           in_Anlage_ein            := #iSystemActive,
           in_Quitt_Stoerung        := #aFBRotaryValve,
           in_Ansteuerung_Motor     := #RotaryFeeder.auto_mode_control,
           in_Eingang_Motor         := #iFBRotaryFeeder_on,
           io_Ausgang_Motor         := #qRotaryValve_on,
           io_Motor_in_Betrieb      := #RotaryFeeder.motor_in_operation,
           io_Stoerung              := #fFBRotaryFeeder,
           io_Motorstruktur         := #RotaryFeeder);
NETWORK
TITLE = Discharging: release filter
      A     #SEQUENCE.Discharging.AUTO;
      A     #SEQUENCE.Discharging.RELEASE;
      A     #RotaryFeeder.motor_in_operation;
      AN    #PurgedFilter.auto_mode_control_clock1;
      =     #PurgedFilter.auto_mode_control_clock2;
NETWORK
TITLE = Air purge filter object
      CALL  "FC23 Valve 1-10O" (
           in_Handbedienung_erlaubt := TRUE,
           in_Anlage_ein            := #iSystemActive,
           in_Ansteuerung_Ventil_T1 := #PurgedFilter.auto_mode_control_clock1,
           in_Ansteuerung_Ventil_T2 := #PurgedFilter.auto_mode_control_clock2,
           io_Ausgang_Ventil_1      := #qPurgingFilterV1_on,
           io_Ausgang_Ventil_2      := #qPurgingFilterV2_on,
           io_Ausgang_Ventil_3      := #qPurgingFilterV3_on,
           io_Ausgang_Ventil_4      := #PurgedFilter.quit_valve_5,
           io_Ausgang_Ventil_5      := #PurgedFilter.quit_valve_5,
           io_Ausgang_Ventil_6      := #PurgedFilter.quit_valve_6,
           io_Ausgang_Ventil_7      := #PurgedFilter.quit_valve_7,
           io_Ausgang_Ventil_8      := #PurgedFilter.quit_valve_8,
           io_Ausgang_Ventil_9      := #PurgedFilter.quit_valve_9,
           io_Ausgang_Ventil_10     := #PurgedFilter.quit_valve_10,
           io_Ventil_in_Betrieb     := #PurgedFilter.valve_in_operation,
           io_Ventilstruktur        := #PurgedFilter);
NETWORK
TITLE = Discharging: DISCHARGING ACTIVE
      A     #SEQUENCE.Discharging.RELEASE;
      A     #RotaryFeeder.motor_in_operation;
      A     #Screener.motor_in_operation;
      A     #MetalSeparator.motor_in_operation;
      =     #SEQUENCE.Discharging.ACTIVE;
NETWORK
TITLE = -----------PFCs---------------
NETWORK
TITLE = PFCs: PFC to packing Machine
      A     #SEQUENCE.Discharging.ACTIVE;	// system is ON + feeding is started
      AN    #fRepRotaryValve;
      AN    #fRepScreener;
      AN    #fRepMetalSeparator;
      AN    #fFBRotaryFeeder;
      AN    #fFBScreener;
      AN    #fFBMetalSeparator;
      AN    #fSafetyRotaryFeeder;
      AN    #fToolKeyControl;
      AN    #fSafetyMS;
      AN    #fREC01HighLevel;
      =     #qPFCPM_Active;
      O     #INTERNAL.Flags.StatusHP03.HP03_material_signal;
      O     #INTERNAL.Flags.StatusREC01.REC01_material_signal;
      =     #qPFCPM_Product;
NETWORK
TITLE = ---------Statuses to HMI----------------
NETWORK
TITLE = Status to HMI: Filling STATUS
      AN    #SEQUENCE.Filling.RELEASE;
      AN    #SEQUENCE.Filling.ACTIVE;
      JCN   FRA;	// status release assignment
      L     0;
      JU    FAF;	// status assignmnet is finished 
FRA:  A     #SEQUENCE.Filling.RELEASE;
      AN    #SEQUENCE.Filling.ACTIVE;
      JCN   FAA;	// status active 
      L     1;
      JU    FAF;
FAA:  A     #SEQUENCE.Filling.RELEASE;
      A     #SEQUENCE.Filling.ACTIVE;
      L     2;
FAF:  T     #HMI.PV.StatusProcessFilling;
NETWORK
TITLE = Status to HMI: Discharging STATUS
      AN    #SEQUENCE.Discharging.RELEASE;
      AN    #SEQUENCE.Discharging.ACTIVE;
      JCN   DRA;	// status release assignment
      L     0;
      JU    DAF;	// status assignmnet is finished 
DRA:  A     #SEQUENCE.Discharging.RELEASE;
      AN    #SEQUENCE.Discharging.ACTIVE;
      JCN   DAA;	// status active 
      L     1;
      JU    DAF;
DAA:  A     #SEQUENCE.Discharging.RELEASE;
      A     #SEQUENCE.Discharging.ACTIVE;
      L     2;
DAF:  T     #HMI.PV.StatusProcessDischarging;
NETWORK
TITLE = Statuses to HMI for REC01 and HP03 
      A     #INTERNAL.Flags.StatusREC01.REC01_empty;
      =     #HMI.STATE.REC01_empty;
      A     #INTERNAL.Flags.StatusREC01.REC01_full;
      =     #HMI.STATE.REC01_full;
      A     #INTERNAL.Flags.StatusREC01.REC01_material_signal;
      =     #HMI.STATE.REC01_material_signal;
      A     #INTERNAL.Flags.StatusHP03.HP03_empty;
      =     #HMI.STATE.HP03_empty;
      A     #INTERNAL.Flags.StatusHP03.HP03_full;
      =     #HMI.STATE.HP03_full;
      A     #INTERNAL.Flags.StatusHP03.HP03_material_signal;
      =     #HMI.STATE.HP03_material_signal;
NETWORK
TITLE = Status to HMI: PFC to/from Rovema 
//from Rovema
      A     #iPFCPM_Ready;
      =     #HMI.STATE.FROMRovemaReady;
      A     #iPFCPM_TakeProduct;
      =     #HMI.STATE.FROMRovemaTakeMaterial;
// to Rovema
      A     #qPFCPM_Product;
      =     #HMI.STATE.TORovemaProductHP03;
      A     #qPFCPM_Active;
      =     #HMI.STATE.TORovemaActive;
NETWORK
TITLE = ------------Resetting----------------
NETWORK
TITLE = Reset Storage Location
      O     #INTERNAL.Flags.ReleaseFeeding;
      O     #INTERNAL.Flags.StatusREC01.REC01_material_signal;
      O     #INTERNAL.Flags.StatusHP03.HP03_material_signal;
      ON    #iSystemActive;
      FP    #INTERNAL.Flags.FP_StorageLocReset.helpBit;
      =     #INTERNAL.Flags.FP_StorageLocReset.pulseBit;
      A     #INTERNAL.Flags.FP_StorageLocReset.pulseBit;
      JCN   NRS;	//no reset storage
      L     0;
      T     #HMI.PARAM.StorageLocation;
NRS:  NOP   0;
NETWORK
TITLE = ---- interface ----
NETWORK
TITLE = Storage location
      A     #iSystemActive;
      A     #INTERNAL.IF.Silo.SiloNr_correct;
      JCN   NCS;	// correst silo number
      L     #HMI.PV.StorageLocation;
      L     1000;
      +I;
      T     #INTERNAL.IF.Silo.StorageLocation_DB;
      L     200;
      T     #INTERNAL.IF.Silo.StorageLocation_DW;
      CALL  "FC40 copy Obj-IF Master" (
           i_Freigabe               := #IF_Silo.CONTROL.CMD.Request,
           i_Ziel_DB                := #INTERNAL.IF.Silo.StorageLocation_DB,
           i_Ziel_DW                := #INTERNAL.IF.Silo.StorageLocation_DW,
           i_SST_von_Ziel           := #IF_Silo.STATUS,
           i_SST_an_Ziel            := #IF_Silo.CONTROL,
           Ziel_frei                := #INTERNAL.IF.Silo.Silo_free);
NCS:  NOP   0;
NETWORK
TITLE = Blower
      L     #IF_Blower_DB;
      T     #INTERNAL.IF.Blower.Blower_DB;
      L     #IF_Blower_DW;
      T     #INTERNAL.IF.Blower.Blower_DW;
      CALL  "FC40 copy Obj-IF Master" (
           i_Freigabe               := #IF_Blower.CONTROL.CMD.Request,
           i_Ziel_DB                := #INTERNAL.IF.Blower.Blower_DB,
           i_Ziel_DW                := #INTERNAL.IF.Blower.Blower_DW,
           i_SST_von_Ziel           := #IF_Blower.STATUS,
           i_SST_an_Ziel            := #IF_Blower.CONTROL,
           Ziel_frei                := #INTERNAL.IF.Blower.Blower_free);
NETWORK
TITLE = -----------Signals to Rovema--------------
NETWORK
TITLE = Discharging: ready signal to packing machine
      A     #SEQUENCE.Discharging.AUTO;
      AN    #fRepRotaryValve;
      AN    #fRepScreener;
      AN    #fRepMetalSeparator;
      AN    #fSafetyRotaryFeeder;
      A     #INTERNAL.IF.Silo.SiloNr_correct;
      =     #qPFCPM_Product;
END_FUNCTION_BLOCK

FUNCTION_BLOCK "PMP01"	// FB 1051
TITLE = Blower PMP01
//Creation:
//Date:            Author:                                               Version
//--------------------------------------------------------------------------------
//18.04.2017      Ilia Bedniakov (ilia)                                  01.00.00
//
//Changes:
//No. Date:        Who       Description                           Mark   Version 
//--------------------------------------------------------------------------------
//01
//________________________________________________________________________________
//Function:
//
VERSION : 0.1
VAR_INPUT
  piwPressure : INT ;	//analogue input address
  SystemActive : BOOL ;	//system on
  iFBBlower_on : BOOL ;
  iRepBlower_on : BOOL ;
  aFBBlower : BOOL ;	//ack feedback fault
  aRepBlower : BOOL ;	//ack repair switch fault
END_VAR
VAR_IN_OUT
  qBlower_on : BOOL ;
  fFBBlower : BOOL ;	//feedback fault
  fRepBlower : BOOL ;	//repair switch fault
  fPressureFault : BOOL ;	//fault pressure value
  wBrokenWirePT : BOOL ;	//wire break fault
END_VAR
VAR
  reserve_IO : ARRAY  [6 .. 49 ] OF BYTE ;
  HMI : STRUCT 	//Interface of HMI
   CMD : STRUCT
    reserve : BOOL ;
    reserve_1 : BOOL ;
    reserve_2 : BOOL ;
    reserve_3 : BOOL ;
    reserve_4 : BOOL ;
    reserve_5 : BOOL ;
    reserve_6 : BOOL ;
    reserve_7 : BOOL ;
    reserve_8 : BOOL ;
    reserve_9 : BOOL ;
    reserve_10 : BOOL ;
    reserve_11 : BOOL ;
    reserve_12 : BOOL ;
    reserve_13 : BOOL ;
    reserve_14 : BOOL ;
    reserve_15 : BOOL ;
   END_STRUCT ;
   STATE : STRUCT
    BlowerLocked : BOOL ;
    PressureFault : BOOL ;
    reserve : BOOL ;
    reserve_1 : BOOL ;
    reserve_2 : BOOL ;
    reserve_3 : BOOL ;
    reserve_4 : BOOL ;
    reserve_5 : BOOL ;
    reserve_6 : BOOL ;
    reserve_7 : BOOL ;
    reserve_8 : BOOL ;
    reserve_9 : BOOL ;
    reserve_10 : BOOL ;
    reserve_11 : BOOL ;
    reserve_12 : BOOL ;
    reserve_13 : BOOL ;
   END_STRUCT ;
   PARAM : STRUCT
    BlowerOffDelayTime : REAL  := 1.000000e+001;
    MinPressure : REAL  := -3.000000e+002;
    MaxPressure : REAL  := -5.000000e+002;
    EmptyPressure : REAL  := -2.000000e+002;
    BlockStart : REAL  := 3.000000e+002;
    reserve : REAL ;
    reserve_1 : REAL ;
    reserve_2 : REAL ;
    reserve_3 : REAL ;
    reserve_4 : INT ;
    reserve_5 : INT ;
    reserve_6 : INT ;
    reserve_7 : INT ;
    reserve_8 : INT ;
    reserve_9 : INT ;
   END_STRUCT ;
   PV : STRUCT
    BlowerOffDelayTime : REAL ;
    ActualPressure : REAL ;
    BlowerRestarInterval : REAL ;
    reserve : REAL ;
    reserve_1 : REAL ;
    reserve_2 : REAL ;
    reserve_3 : REAL ;
    reserve_4 : REAL ;
    reserve_5 : INT ;
    reserve_6 : INT ;
    reserve_7 : INT ;
    reserve_8 : INT ;
    reserve_9 : INT ;
    reserve_10 : INT ;
    reserve_11 : INT ;
    reserve_12 : INT ;
   END_STRUCT ;
  END_STRUCT ;
  PROD : STRUCT 	//Interface of Production
   FROM : STRUCT
    reserve : INT ;
    reserve_1 : INT ;
    reserve_2 : INT ;
    reserve_3 : INT ;
    reserve_4 : INT ;
    reserve_5 : REAL ;
    reserve_6 : REAL ;
    CMD : STRUCT
     reserve : BOOL ;
     reserve_1 : BOOL ;
     reserve_2 : BOOL ;
     reserve_3 : BOOL ;
     reserve_4 : BOOL ;
     reserve_5 : BOOL ;
     reserve_6 : BOOL ;
     reserve_7 : BOOL ;
     reserve_8 : BOOL ;
     reserve_9 : BOOL ;
     reserve_10 : BOOL ;
     reserve_11 : BOOL ;
     reserve_12 : BOOL ;
     reserve_13 : BOOL ;
     reserve_14 : BOOL ;
     reserve_15 : BOOL ;
    END_STRUCT ;
   END_STRUCT ;
   TO : STRUCT
    reserve : INT ;
    reserve_1 : INT ;
    reserve_2 : INT ;
    reserve_3 : INT ;
    reserve_4 : INT ;
    reserve_5 : REAL ;
    reserve_6 : REAL ;
    STATE : STRUCT
     reserve : BOOL ;
     reserve_1 : BOOL ;
     reserve_2 : BOOL ;
     reserve_3 : BOOL ;
     reserve_4 : BOOL ;
     reserve_5 : BOOL ;
     reserve_6 : BOOL ;
     reserve_7 : BOOL ;
     reserve_8 : BOOL ;
     reserve_9 : BOOL ;
     reserve_10 : BOOL ;
     reserve_11 : BOOL ;
     reserve_12 : BOOL ;
     reserve_13 : BOOL ;
     reserve_14 : BOOL ;
     reserve_15 : BOOL ;
    END_STRUCT ;
   END_STRUCT ;
   reserve : ARRAY  [40 .. 49 ] OF BYTE ;
  END_STRUCT ;
  IF_Consumer : STRUCT 	//Interface Blower in blower object
   CONTROL : STRUCT
    Answer_DB : INT ;
    Answer_DW : INT ;
    reserve_1 : INT ;
    reserve_2 : INT ;
    reserve_3 : INT ;
    reserve_4 : REAL ;
    reserve_5 : REAL ;
    CMD : STRUCT
     Request : BOOL ;
     Release : BOOL ;
     EmergencyStopBlower : BOOL ;
     reserve : BOOL ;
     reserve_1 : BOOL ;
     reserve_2 : BOOL ;
     reserve_3 : BOOL ;
     reserve_4 : BOOL ;
     reserve_5 : BOOL ;
     reserve_6 : BOOL ;
     reserve_7 : BOOL ;
     reserve_8 : BOOL ;
     reserve_9 : BOOL ;
     reserve_10 : BOOL ;
     reserve_11 : BOOL ;
     DataExchange : BOOL ;
    END_STRUCT ;
   END_STRUCT ;
   STATE : STRUCT
    reserve_1 : INT ;
    reserve_2 : INT ;
    reserve_3 : INT ;
    reserve_4 : INT ;
    reserve_5 : INT ;
    reserve_6 : REAL ;
    reserve_7 : REAL ;
    STATE : STRUCT
     Ready : BOOL ;
     Active : BOOL ;
     PressureFault : BOOL ;
     EmptyPressurReached : BOOL ;
     reserve : BOOL ;
     reserve_1 : BOOL ;
     reserve_2 : BOOL ;
     reserve_3 : BOOL ;
     reserve_4 : BOOL ;
     reserve_5 : BOOL ;
     reserve_6 : BOOL ;
     reserve_7 : BOOL ;
     reserve_8 : BOOL ;
     reserve_9 : BOOL ;
     reserve_10 : BOOL ;
     reserve_11 : BOOL ;
    END_STRUCT ;
   END_STRUCT ;
  END_STRUCT ;
  reserve_IF : ARRAY  [240 .. 499 ] OF BYTE ;
  Blower : STRUCT 	//motor object
   parameter : STRUCT
    motor_on : BOOL  := TRUE;	//activate motor structure
    clock_on : BOOL ;	//activate clock structure
    FC_on : BOOL ;	//activate frequency converter structure
    hour_meter_on : BOOL ;	//activate hour meter
    reserve_4 : BOOL ;
    reserve_5 : BOOL ;
    reserve_6 : BOOL ;
    reserve_7 : BOOL ;
   END_STRUCT ;
   quit_motor : BOOL ;	//1 = quit motor on
   input_motor : BOOL ;	//1 = input motor on (return indication)
   motor_locked : BOOL ;	//1 = motor locked (in manual and auto mode) e.g. repair-/safety switch
   auto_mode_control : BOOL ;	//1 = release/control of motor in auto mode
   motor_in_operation : BOOL ;	//1 = signal motor in operation
   fault : BOOL ;	//1 = signal motor fault
   man_mode_to_SCADA : BOOL ;	//0 = Automatik Mode, 1 = Hand Mode
   man_mode_from_SCADA : BOOL ;	//0 = Automatik Mode, 1 = Hand Mode
   man_mode_control : BOOL ;	//1 = release/control of motor in manual mode (from SCADA)
   man_mode_locked : BOOL ;	//1 = change to manual mode locked, motor is in automatic use
   start_with_impulse : BOOL  := TRUE;	//1 = start cycle with impulse
   set_cycles_reached : BOOL ;	//1 = set number of cycles has been reached
   continous_clock : BOOL  := TRUE;	//1 = continous clock / 0 = set number of clocks
   simulation : BOOL ;	//1 = simulation of object
   release_clock : BOOL ;	//1 = release bit for clock FC
   quit_clock : BOOL ;	//quit for clock FC, if release_clock = TRUE
   set_time_fault : INT  := 5;	//fault evaluation time in seconds
   actual_time_fault : INT ;	//actual fault evaluation time in seconds
   impulse_time : REAL  := 5.000000e+000;	//impulse time for clock in seconds
   break_time : REAL  := 5.000000e+000;	//break time for clock in seconds
   time_counter : REAL ;	//time counter (elapsed time)
   set_cycles : INT ;	//number of clocks if not continous clock
   clock_counter : INT ;	//clock counter
   FCs : STRUCT 	//frequency converter
    FC_in_operation : BOOL ;	//1 = FU in Betrieb
    fault : BOOL ;	//1 = FC fault
    set_revolutions_man_mode : INT ;	//revolutions in permille in manual mode
    actual_revolutions : INT ;	//actual revolutions FC in man/auto mode
   END_STRUCT ;
   hour_meter : STRUCT 	//hour meter
    reset : BOOL ;	//reset hour meter
    warning : BOOL ;	//warning time exceeded
    alarm : BOOL ;	//alarm time exceeded
    actual_operating_hours : REAL ;	//actual operating hours (in hours)
    set_time_warning : REAL ;	//set time for warning (in hours)
    set_time_alarm : REAL ;	//set time for alarm (in hours)
    second_counter_oh : INT ;	//seconds of the actual operatin hours
   END_STRUCT ;
   system_on : BOOL ;	//system released resepectively system area released after emergency stopping
   object_state : INT ;	//1=grey; 5=green; 9=white; 15=yellow; 16=red
  END_STRUCT ;
  reserve_Cmod : ARRAY  [600 .. 999 ] OF BYTE ;
  TIMES : STRUCT 	//ten timers
   TOF_Blower : STRUCT
    IN : BOOL ;
    RST : BOOL ;
    IMP : BOOL ;
    Q : BOOL ;
    PT : REAL ;
    ET : REAL ;
   END_STRUCT ;
   TOF_BlowerRestarInterval : STRUCT
    IN : BOOL ;
    RST : BOOL ;
    IMP : BOOL ;
    Q : BOOL ;
    PT : REAL ;
    ET : REAL ;
   END_STRUCT ;
   reserve : STRUCT
    IN : BOOL ;
    RST : BOOL ;
    IMP : BOOL ;
    Q : BOOL ;
    PT : REAL ;
    ET : REAL ;
   END_STRUCT ;
   reserve_1 : STRUCT
    IN : BOOL ;
    RST : BOOL ;
    IMP : BOOL ;
    Q : BOOL ;
    PT : REAL ;
    ET : REAL ;
   END_STRUCT ;
   reserve_2 : STRUCT
    IN : BOOL ;
    RST : BOOL ;
    IMP : BOOL ;
    Q : BOOL ;
    PT : REAL ;
    ET : REAL ;
   END_STRUCT ;
   reserve_3 : STRUCT
    IN : BOOL ;
    RST : BOOL ;
    IMP : BOOL ;
    Q : BOOL ;
    PT : REAL ;
    ET : REAL ;
   END_STRUCT ;
   reserve_4 : STRUCT
    IN : BOOL ;
    RST : BOOL ;
    IMP : BOOL ;
    Q : BOOL ;
    PT : REAL ;
    ET : REAL ;
   END_STRUCT ;
   reserve_5 : STRUCT
    IN : BOOL ;
    RST : BOOL ;
    IMP : BOOL ;
    Q : BOOL ;
    PT : REAL ;
    ET : REAL ;
   END_STRUCT ;
  END_STRUCT ;
  SEQUENCES : STRUCT
   Sequence : STRUCT
    AUTO : BOOL ;
    MANUAL : BOOL ;
    LOCKED : BOOL ;
    reserve : BOOL ;
    reserve_1 : BOOL ;
    reserve_2 : BOOL ;
    reserve_3 : BOOL ;
    reserve_4 : BOOL ;
    reserve_5 : BOOL ;
    reserve_6 : BOOL ;
    reserve_7 : BOOL ;
    reserve_8 : BOOL ;
    reserve_9 : BOOL ;
    reserve_10 : BOOL ;
    reserve_11 : BOOL ;
    reserve_12 : BOOL ;
   END_STRUCT ;
   reserve : ARRAY  [2 .. 99 ] OF BYTE ;
  END_STRUCT ;
  INTERNAL : STRUCT
   IF : STRUCT
    reserve : BOOL ;
    reserve_1 : BOOL ;
    reserve_2 : BOOL ;
    reserve_3 : BOOL ;
    reserve_4 : BOOL ;
    reserve_5 : BOOL ;
    reserve_6 : BOOL ;
    reserve_7 : BOOL ;
    reserve_8 : BOOL ;
    reserve_9 : BOOL ;
    reserve_10 : BOOL ;
    reserve_11 : BOOL ;
    reserve_12 : BOOL ;
    reserve_13 : BOOL ;
    reserve_14 : BOOL ;
    reserve_15 : BOOL ;
   END_STRUCT ;
   Flags : STRUCT
    FP_Blower_on : BOOL ;
    reserve : BOOL ;
    reserve_1 : BOOL ;
    reserve_2 : BOOL ;
    reserve_3 : BOOL ;
    reserve_4 : BOOL ;
    reserve_5 : BOOL ;
    reserve_6 : BOOL ;
    reserve_7 : BOOL ;
    reserve_8 : BOOL ;
    reserve_9 : BOOL ;
    reserve_10 : BOOL ;
    reserve_11 : BOOL ;
    reserve_12 : BOOL ;
    reserve_13 : BOOL ;
   END_STRUCT ;
   PressureTransmitter : STRUCT
    Analog : STRUCT
     in : STRUCT
      UperLimit : REAL  := 1.000000e+003;	//Uper limit analog value
      LowerLimit : REAL  := -1.000000e+003;	//Lower limit analog value
      MaxDigit : REAL  := 2.764800e+004;	//Uper limit analog channel
      MinDigit : REAL ;	//Lower limit analog channel
      Simulation : BOOL ;	//Simulation = 1
      DB_Simulation_IO : INT  := 92;	//DB for simulation
     END_STRUCT ;
     out : STRUCT
      Value : REAL ;	//IO Analog value
      Broken_wire : BOOL ;	//Fault broken wire
      Reserve : INT ;
     END_STRUCT ;
    END_STRUCT ;
    Evaluation : STRUCT
     in : STRUCT
      Delay_Adjust : REAL  := 1.000000e+001;	//Delay adjust of Pressure Transmitter
      Selection_S_D : CHAR  := 'S';	//Selection suction-/pressure conveying ('S' or 'D')
      REL_Pressure_fault : BOOL  := TRUE;	//Release Pressure fault
      Time_counter : REAL ;	//Time counter delay adjust
      Output_Timer : BOOL ;	//Timer output delay adjust
     END_STRUCT ;
     out : STRUCT
      Relative_Pressure : REAL ;	//Relative Pressure
      Memory_Pressure : REAL ;	//Memory Pressure
      Pressure_fault_active : BOOL ;	//Pressure fault
      Empty_Pressure_reached : BOOL ;	//Below Empty Pressure
      output_delay_calibration : BOOL ;
     END_STRUCT ;
    END_STRUCT ;
   END_STRUCT ;
   Instance_DB_number : INT ;
  END_STRUCT ;
END_VAR
BEGIN
NETWORK
TITLE = ---- instance DB ----
      L     0;
      L     DINO;
      ==I;
      BEC;
      T     #INTERNAL.Instance_DB_number;
NETWORK
TITLE = ---- Sequence status ----
NETWORK
TITLE =  Sequence Auto
      O     #IF_Consumer.CONTROL.CMD.Request;
      O     #TIMES.TOF_Blower.Q;
      AN    #SEQUENCES.Sequence.LOCKED;
      =     #SEQUENCES.Sequence.AUTO;
NETWORK
TITLE =  Sequence Manual
      O     #Blower.man_mode_to_SCADA;
      AN    #SEQUENCES.Sequence.AUTO;
      =     #SEQUENCES.Sequence.MANUAL;
NETWORK
TITLE =  Sequence Locked
      ON    #SystemActive;
      O     #SEQUENCES.Sequence.MANUAL;
      =     #SEQUENCES.Sequence.LOCKED;
NETWORK
TITLE = ----General module ----
NETWORK
TITLE = blower repair switch
      A     #iRepBlower_on;
      A     #aRepBlower;
      R     #fRepBlower;
      O     #Blower.auto_mode_control;
      O     #Blower.man_mode_control;
      AN    #iRepBlower_on;
      S     #fRepBlower;
NETWORK
TITLE = pressure trassmitter 
//pressure read
      CALL  "FC10 Analogue value r/w" (
           in_E_A                   := B#16#45,
           in_EA_Adresse            := #piwPressure,
           in_OberGrenze            := 1.000000e+03,
           in_UnterGrenze           := -1.000000e+03,
           in_MaxDigit              := 2.764800e+04,
           in_MinDigit              := 0.000000e+00,
           in_Typ                   := B#16#5A,
           in_Simulation            := "M 0.5 InternalSimulation",
           in_DB_Simulation_EA      := 32,
           io_Wert                  := #INTERNAL.PressureTransmitter.Analog.out.Value,
           io_Drahtbruch            := #INTERNAL.PressureTransmitter.Analog.out.Broken_wire);
      A     #INTERNAL.PressureTransmitter.Analog.out.Broken_wire;
      =     #wBrokenWirePT;
//pressure evaluation
      CALL  "FC11 PressureTransmitter" (
           AbsolutDruck             := #INTERNAL.PressureTransmitter.Analog.out.Value,
           MinDruck                 := #HMI.PARAM.MinPressure,
           MaxDruck                 := #HMI.PARAM.MaxPressure,
           LeerDruck                := #HMI.PARAM.EmptyPressure,
           Verz_Abgleich            := 1.800000e+02,
           Auswahl_S_D              := B#16#53,
           Drahtbruch               := #INTERNAL.PressureTransmitter.Analog.out.Broken_wire,
           Geblaese_aktiv           := #qBlower_on,
           FRG_Druckstoerung        := #INTERNAL.PressureTransmitter.Evaluation.in.REL_Pressure_fault,
           Zeitzaehler              := #INTERNAL.PressureTransmitter.Evaluation.in.Time_counter,
           RelativDruck             := #INTERNAL.PressureTransmitter.Evaluation.out.Relative_Pressure,
           MemoryDruck              := #INTERNAL.PressureTransmitter.Evaluation.out.Memory_Pressure,
           Druckstoerung            := #INTERNAL.PressureTransmitter.Evaluation.out.Pressure_fault_active,
           Leerdruck_aktiv          := #INTERNAL.PressureTransmitter.Evaluation.out.Empty_Pressure_reached,
           Ausgang_Timer            := #INTERNAL.PressureTransmitter.Evaluation.out.output_delay_calibration);	// No Frishluft Ventile /  Vacuum Pump
      L     #INTERNAL.PressureTransmitter.Evaluation.out.Relative_Pressure;
      T     #HMI.PV.ActualPressure;
NETWORK
TITLE = ---- Sequence ----
NETWORK
TITLE = Sequence: ready to consumer
      A     #SEQUENCES.Sequence.AUTO;
      A     #IF_Consumer.CONTROL.CMD.Request;
      =     #IF_Consumer.STATE.STATE.Ready;
NETWORK
TITLE = Sequence: release blower 
//blower off delay
      A     #SEQUENCES.Sequence.AUTO;
      A     #IF_Consumer.STATE.STATE.Ready;
      A     #IF_Consumer.CONTROL.CMD.Release;
      AN    #IF_Consumer.CONTROL.CMD.EmergencyStopBlower;
      =     #TIMES.TOF_Blower.IN;
      ON    #SystemActive;
      O     #Blower.man_mode_to_SCADA;
      O     #IF_Consumer.CONTROL.CMD.EmergencyStopBlower;
      =     #TIMES.TOF_Blower.RST;
      CALL  "FC3 Cycle generator" (
           in_Freigabe              := #TIMES.TOF_Blower.IN,
           in_Reset                 := #TIMES.TOF_Blower.RST,
           in_Impuls                := "M 1.7 Cycle Timer-FC",
           in_Impulszeit_in_100ms   := "MW 6 Timer Val Cycle FCs",
           in_Verzoegerungsart      := B#16#41,
           in_Verzoegerungszeit     := #HMI.PARAM.BlowerOffDelayTime,
           io_Ausgangssignal        := #TIMES.TOF_Blower.Q,
           io_Zeitzaehler           := #TIMES.TOF_Blower.ET);
      L     #TIMES.TOF_Blower.ET;
      T     #HMI.PV.BlowerOffDelayTime;
NETWORK
TITLE = Block next start
//restart protection 
      A     #qBlower_on;
      FP    #INTERNAL.Flags.FP_Blower_on;
      =     #TIMES.TOF_BlowerRestarInterval.IN;
//only 12 times per hour 
      CALL  "FC3 Cycle generator" (
           in_Freigabe              := #TIMES.TOF_BlowerRestarInterval.IN,
           in_Reset                 := FALSE,
           in_Impuls                := "M 1.7 Cycle Timer-FC",
           in_Impulszeit_in_100ms   := "MW 6 Timer Val Cycle FCs",
           in_Verzoegerungsart      := B#16#41,
           in_Verzoegerungszeit     := #HMI.PARAM.BlockStart,
           io_Ausgangssignal        := #TIMES.TOF_BlowerRestarInterval.Q,
           io_Zeitzaehler           := #TIMES.TOF_BlowerRestarInterval.ET);
      L     #TIMES.TOF_BlowerRestarInterval.ET;
      T     #HMI.PV.BlowerRestarInterval;
NETWORK
TITLE = Blower Motor object
//release blower
      A     #SEQUENCES.Sequence.AUTO;
      A     #TIMES.TOF_Blower.Q;
      =     #Blower.auto_mode_control;
      A     #SEQUENCES.Sequence.AUTO;
      AN    "Service mode lock auto";
      =     #Blower.man_mode_locked;
      A     #TIMES.TOF_BlowerRestarInterval.Q;
      AN    #qBlower_on;
      O     #fRepBlower;
      ON    #iRepBlower_on;
      =     #Blower.motor_locked;
      A     #Blower.motor_locked;
      =     #HMI.STATE.BlowerLocked;
      CALL  "FC20 Motor 1O1I" (
           in_Handbedienung_erlaubt := TRUE,
           in_Quitt_Stoerung_noetig := TRUE,
           in_Anlage_ein            := #SystemActive,
           in_Quitt_Stoerung        := #aFBBlower,
           in_Ansteuerung_Motor     := #Blower.auto_mode_control,
           in_Eingang_Motor         := #iFBBlower_on,
           io_Ausgang_Motor         := #qBlower_on,
           io_Motor_in_Betrieb      := #Blower.motor_in_operation,
           io_Stoerung              := #fFBBlower,
           io_Motorstruktur         := #Blower);
NETWORK
TITLE = Sequence: active to consumer
      A     #SEQUENCES.Sequence.AUTO;
      A     #IF_Consumer.CONTROL.CMD.Release;
      A     #Blower.motor_in_operation;
      =     #IF_Consumer.STATE.STATE.Active;
//pressure fault
      A     #INTERNAL.PressureTransmitter.Evaluation.out.Pressure_fault_active;
      =     #IF_Consumer.STATE.STATE.PressureFault;
      =     #fPressureFault;
      =     #HMI.STATE.PressureFault;
//emty pressure reached
      A     #INTERNAL.PressureTransmitter.Evaluation.out.Empty_Pressure_reached;
      =     #IF_Consumer.STATE.STATE.EmptyPressurReached;
NETWORK
TITLE = ---- Interface ----
NETWORK
TITLE = interface Consumer
      CALL  "FC41 copy Obj-IF Slave" (
           i_SST_von_Ziel           := #IF_Consumer.CONTROL,
           i_SST_an_Ziel            := #IF_Consumer.STATE);
END_FUNCTION_BLOCK

FUNCTION_BLOCK "FC01_RV_HOPPERS"	// FB 4901
TITLE = FU Auswahlbaustein
//Erstellung:
//Datum        Bearbeiter                                                 Version
//--------------------------------------------------------------------------------
//10.07.06     Dominik Ilzhöfer (id)                                      01.00.00
//
//Änderungen:
//Nr. Datum    Bearb Änderung                                       Marke  Version
//--------------------------------------------------------------------------------
//01  06.11.07 sra   Motornennfrequenz und Motornenndrehzahl eingef.(001) 01.01.00
//02  23.07.13 sra   Status FU eingefügt                            (002) 01.02.00
//
//Baustein zur Ansteuerung von Frequenzumformern über Profibus-DB
//
//Parametrierung:
//FU-Typ:        wird zur richtigen Fehleranzeige an der Visualisierung benötigt
//               1=Siemens-MM4
//               2=SEW UFP11A
//               3=Lenze E82ZAFPC
//               4=Danfoss VLT5000
//               5=Danfoss FC300
//               6=SEW DFP21B
//             
//PEA-Adresse:   Anfangsadresse der Profibus-Schnittstelle
//Motordaten-DB: DB-Nummer mit Motordaten (Standard = DB4)
//FU-Nummer    : wird nur bei SEW Frequenzumformern mit UFP11A und DFP21B benötigt
//
//!Achtung!
//Bei den SEW Frequenzumformern wird die Motornennfrequenz und die 
//Motornenndrehzahl benötigt. D.h. es muss entweder ein Motordatensatz in dem 
//Motordaten-DB vorhanden sein oder die Werte müssen dem Baustein übergeben 
//werden.
VERSION : 0.1
VAR_INPUT
  in_FU_Typ : INT ;	//1=Siemens-MM4, 2=SEW UFP11A, 3=Lenze E82ZAFPC, 4=Danfoss VLT5000
  in_PEA_Adresse : INT ;	//Basisadresse für EA-Daten im PEA-Bereich
  in_Motordaten_DB : INT  := 1;	//Adresse des DBs für Motordaten ( 0 = keine Motordaten schreiben )
  in_FU_Nummer : INT ;	//Nummer des FUs (für SEW-FUs)
  in_Motornennfrequenz : REAL ;	//muss bei SEW-FUs angegeben werden wenn kein Motordatensatz vorhanden ist
  in_Motornenndrehzahl : REAL ;	//muss bei SEW-FUs angegeben werden wenn kein Motordatensatz vorhanden ist
END_VAR
VAR_IN_OUT
  FU_Stoerung : BOOL ;
END_VAR
VAR
  reserve : ARRAY  [18 .. 29 ] OF BYTE ;
  Daten_Visualisierung : STRUCT
   von : STRUCT
    Quittierung_Stoerung : BOOL ;
    reserve : ARRAY  [2 .. 19 ] OF BYTE ;
   END_STRUCT ;
   an : STRUCT
    FU_Typ : INT ;
    Freigabe : BOOL ;
    Laeuft : BOOL ;
    Stoerung : BOOL ;
    Warnung : BOOL ;
    Sollfrequenz_erreicht : BOOL ;
    Sollfrequenz : REAL ;
    Istfrequenz : REAL ;
    Istdrehzahl : REAL ;
    Ausgangsstrom : REAL ;
    Leistung : REAL ;
    Drehmoment : REAL ;
    Spannung : REAL ;
    FU_Nummer : INT ;
    FB_Fehlermeldung : INT ;
    Stoerungsnummer : DINT ;
    reserve : ARRAY  [40 .. 47 ] OF BYTE ;
    Status : INT ;
   END_STRUCT ;
  END_STRUCT ;
  Schnittstelle : STRUCT
   von : STRUCT
    Antwort_DB : INT ;
    Antwort_DW : INT ;
    Sollfrequenz : REAL ;
    Motordatensatz_Nummer : INT ;
    reserve : ARRAY  [10 .. 17 ] OF BYTE ;
    Steuerbits : STRUCT
     Anforderung : BOOL ;
     Freigabe : BOOL ;
     Linkslauf : BOOL ;
    END_STRUCT ;
   END_STRUCT ;
   an : STRUCT
    Istfrequenz : REAL ;
    reserve : ARRAY  [4 .. 17 ] OF BYTE ;
    Statusbits : STRUCT
     Bereit : BOOL ;
     Laeuft : BOOL ;
     Stoerung : BOOL ;
    END_STRUCT ;
   END_STRUCT ;
  END_STRUCT ;
  Motordaten : STRUCT
   Nennleistugsfaktor : REAL ;
   Nennfrequenz : REAL ;
   Nenndrehzahl : REAL ;
   Nennstrom : REAL ;
   Nennspannung : REAL ;
   Nennleistung : REAL ;
   reserve : ARRAY  [24 .. 29 ] OF BYTE ;
  END_STRUCT ;
  Profibus_FB : FB 4;
END_VAR
VAR_TEMP
  Motordaten_schreiben : BOOL ;
  Motordaten_Transfer_Fehl : INT ;
  Motordaten_Adresse_Quell : INT ;
  Motordaten_Adresse_Ziel : INT ;
END_VAR
BEGIN
NETWORK
TITLE = "Motordaten_schreiben" bilden
//Motordaten werden nur geschrieben, wenn ein Motordaten_DB und eine 
//Motordatensatz_Nummer ungleich 0 angegeben werden
      A(;
      L     #in_Motordaten_DB;
      L     0;
      <>I;
      );
      A(;
      L     #Schnittstelle.von.Motordatensatz_Nummer;
      L     0;
      <>I;
      );
      =     #Motordaten_schreiben;
NETWORK
TITLE = Motordatensatz in Motordaten kopieren
//Kompletter Motordatensatz wird aus Motordaten_DB kopiert
      L     #in_Motornennfrequenz;	// (001)
      T     #Motordaten.Nennfrequenz;	// (001)
      L     #in_Motornenndrehzahl;	// (001)
      T     #Motordaten.Nenndrehzahl;	// (001)
      A     #Motordaten_schreiben;
      JCN   SPR1;
      L     #Schnittstelle.von.Motordatensatz_Nummer;	// Nummer des Datensatzes des Motors
      L     -1;
      +I;
      L     30;	// Länge eines Datensatzes
      *I;
      T     #Motordaten_Adresse_Quell;	// Anfangsadresse des Datensatzes
      L     P##Motordaten;
      SRD   3;
      T     #Motordaten_Adresse_Ziel;
      CALL  "FC5 Block Transfer" (
           Quell_Typ                := B#16#44,
           Quell_DB                 := #in_Motordaten_DB,
           Quell_DW                 := #Motordaten_Adresse_Quell,
           Ziel_Typ                 := B#16#49,
           Ziel_DB                  := 0,
           Ziel_DW                  := #Motordaten_Adresse_Ziel,
           Block_Laenge             := 24,
           outFehler                := #Motordaten_Transfer_Fehl);	// DB mit den Motordatensätzen /  Anfangsadresse des Datensatzes /  nicht verwendet da Ziel_Typ :='I' /  Abhängig vom Motordaten_DB
SPR1: NOP   0;
NETWORK
TITLE = Bei Anforderung "Bereit" bilden
      A     #Schnittstelle.von.Steuerbits.Anforderung;
      =     #Schnittstelle.an.Statusbits.Bereit;
NETWORK
TITLE = Auswahl des FU-Typs
//In der Multiinstanz "Profibus_FB" benötigten FU_Baustein im Datentyp angeben
      CALL  #Profibus_FB (
           in_PEA_Adresse           := #in_PEA_Adresse,
           in_FU_Nummer             := #in_FU_Nummer,
           in_Auswahl_Param_satz_2  := #Motordaten_schreiben,
           in_Freigabe              := #Schnittstelle.von.Steuerbits.Freigabe,
           in_Linkslauf             := #Schnittstelle.von.Steuerbits.Linkslauf,
           in_Quittierung_Stoerung  := #Daten_Visualisierung.von.Quittierung_Stoerung,
           in_Sollfrequenz          := #Schnittstelle.von.Sollfrequenz,
           in_Motorleistungsfaktor  := #Motordaten.Nennleistugsfaktor,
           in_Motornennfrequenz     := #Motordaten.Nennfrequenz,
           in_Motornenndrehzahl     := #Motordaten.Nenndrehzahl,
           in_Motornennstrom        := #Motordaten.Nennstrom,
           in_Motornennspannung     := #Motordaten.Nennspannung,
           in_Motornennleistung     := #Motordaten.Nennleistung,
           out_Istfrequenz          := #Daten_Visualisierung.an.Istfrequenz,
           out_Istdrehzahl          := #Daten_Visualisierung.an.Istdrehzahl,
           out_Leistung             := #Daten_Visualisierung.an.Leistung,
           out_Drehmoment           := #Daten_Visualisierung.an.Drehmoment,
           out_Motorspannung        := #Daten_Visualisierung.an.Spannung,
           out_Ausgangsstrom        := #Daten_Visualisierung.an.Ausgangsstrom,
           out_Stoerung             := #Daten_Visualisierung.an.Stoerung,
           out_Warnung              := #Daten_Visualisierung.an.Warnung,
           out_Sollwert_erreicht    := #Daten_Visualisierung.an.Sollfrequenz_erreicht,
           out_laeuft               := #Daten_Visualisierung.an.Laeuft,
           out_FB_Fehlermeldung     := #Daten_Visualisierung.an.FB_Fehlermeldung,
           out_Stoerungsnummer      := #Daten_Visualisierung.an.Stoerungsnummer);
NETWORK
TITLE = Verknüpfungen von Signalen für Visu und Schnittstelle
      L     #in_FU_Typ;
      T     #Daten_Visualisierung.an.FU_Typ;
      L     #in_FU_Nummer;
      T     #Daten_Visualisierung.an.FU_Nummer;
      A     #Schnittstelle.von.Steuerbits.Freigabe;
      =     #Daten_Visualisierung.an.Freigabe;
      L     #Schnittstelle.von.Sollfrequenz;
      T     #Daten_Visualisierung.an.Sollfrequenz;
      L     #Daten_Visualisierung.an.Istfrequenz;
      T     #Schnittstelle.an.Istfrequenz;
      A     #Daten_Visualisierung.an.Laeuft;
      =     #Schnittstelle.an.Statusbits.Laeuft;
      A     #Daten_Visualisierung.an.Stoerung;
      =     #Schnittstelle.an.Statusbits.Stoerung;
      =     #FU_Stoerung;
NETWORK
TITLE = Sollfrequenz löschen
      A     #Schnittstelle.von.Steuerbits.Freigabe;
      JC    M001;
      L     0;
      T     #Schnittstelle.von.Sollfrequenz;
      CLR;
      =     #Daten_Visualisierung.an.Sollfrequenz_erreicht;
M001: NOP   0;
NETWORK
TITLE = Statusanzeige für Visualisierung
//(002)
      L     16;	// Status Störung
      A     #Daten_Visualisierung.an.Stoerung;
      JC    Stat;
      L     13;	// Status Warnung
      A     #Daten_Visualisierung.an.Warnung;
      JC    Stat;
      L     5;	// Status läuft
      A     #Daten_Visualisierung.an.Laeuft;
      JC    Stat;
      L     1;	// Status aus
Stat: T     #Daten_Visualisierung.an.Status;
NETWORK
TITLE = Schnittstellendaten kopieren
      CALL  "FC41 copy Obj-IF Slave" (
           i_SST_von_Ziel           := #Schnittstelle.von,
           i_SST_an_Ziel            := #Schnittstelle.an);
END_FUNCTION_BLOCK

FUNCTION "FC2 Cycle Gen Timer Emul" : VOID	// FC 2
TITLE = Taktgeber
//Erstellung:
//Datum        Bearbeiter                                                 Version
//--------------------------------------------------------------------------------
//16.12.97     R.Schaffert (sra)                                          01.00.00
//  
//Änderungen:
//Nr. Datum    Bearb Änderung                                       Marke  Version
//--------------------------------------------------------------------------------
//01  09.03.99 sra   Variabler Takteingang                          ()    01.01.00
//02  18.03.99 sra   Fehlerbeseitigung                              ()    01.01.01
//03  01.04.99 jm    Taktzähler auch bei Dauertakt aktiv            ()    01.01.02
//04  14.04.99 sra   Fehlerbeseitigung                              ()    01.01.03
//05  20.12.00 sra   Taktanz.err. rücksetzen bei Dauertakt          ()    01.01.04
//
//________________________________________________________________________________
//Beschreibung:
//
//Diese Funktion generiert ein beliebiges Taktsignal ohne Verwendung eines Timers.
//Es muß ein Impulssignal der Standardimpulse MB4 angelegt werden das über die 
//Taktmerker der CPU und dem Standardbaustein FC13 generiert wird
//Die Zykluszeit muß dabei kleiner sein als das verwendete Taktsignal / 2
//
//Achtung !
//- Am Parameter "in_Rueckmeldung" darf nicht "true" oder "false" angelegt 
//  werden, sondern es muss dem Ausgangssignal "io_Taktausgang" folgen ! 
//- Bei Angabe von z.B. "in_Sollanzahl_Takte" = 5 wird der Parameter 
//  "io_Taktzaehler" von 0..4 hochgezählt
//
AUTHOR : sra
FAMILY : Takt
NAME : Takt_TN
VERSION : 0.0
VAR_INPUT
  in_Freigabe : BOOL ;	//Freigabe Takt
  in_Rueckmeldung : BOOL ;	//Rueckmeldung z.B. Eingang ein
  in_Start_mit_Impuls : BOOL ;	//Takt mit positivem Impuls starten
  in_Dauertakt : BOOL ;	//Dauertakt ? (1=Ja / 0=Nein)
  in_Impuls : BOOL ;	//Impulseingang Takt
  in_Impulszeit_in_100ms : INT ;	//Impulszeit in 100ms
  in_Impulszeit : REAL ;	//Impulszeit fuer Takt in Sekunden
  in_Pausezeit : REAL ;	//Pausezeit fuer Takt in Sekunden
  in_Sollanzahl_Takte : INT ;	//Sollanzahl Takte wenn nicht Dauertakt
END_VAR
VAR_IN_OUT
  io_Taktausgang : BOOL ;	//Taktausgang
  io_Taktanzahl_erreicht : BOOL ;	//Meldung Taktanzahl erreicht
  io_Zeitzaehler : REAL ;	//Zeitzähler (abgelaufene Zeit)
  io_Taktzaehler : INT ;	//Taktzähler
END_VAR
BEGIN
NETWORK
TITLE = Rücksetzen der Zähler und Merker
//Wenn keine Freigabe mehr anliegt werden die in_out Parameter auf 0 gesetzt.
//
      A     #in_Freigabe;
      JC    Strt;
      L     1.000000e-02;
      T     #io_Zeitzaehler;
      L     0;
      T     #io_Taktzaehler;
      SET;
      R     #io_Taktausgang;
      R     #io_Taktanzahl_erreicht;
      BEU;
NETWORK
TITLE = Dauerimpuls oder Dauerpause
Strt: NOP   0;
      L     #in_Impulszeit;
      L     0.000000e+00;
      ==R;
      R     #io_Taktausgang;
      BEC;
      L     #in_Pausezeit;
      L     0.000000e+00;
      ==R;
      S     #io_Taktausgang;
      BEC;
NETWORK
TITLE = Start Takt mit Impuls
//Wenn der Takt mit einem Impuls gestartet werden soll, wird der Ausgang beim 
//Start des Taktes zunächst auf 1 gesetzt.
//Bedingung: Zeitzähler und Taktzähler müssen 0 sein
      A     #in_Freigabe;
      A     #in_Start_mit_Impuls;
      A(;
      A(;
      L     #io_Zeitzaehler;
      L     1.000000e-02;
      ==R;
      );
      A(;
      L     #io_Taktzaehler;
      L     0;
      ==I;
      );
      O;
      A     #in_Dauertakt;
      A     #io_Taktanzahl_erreicht;
      );
      S     #io_Taktausgang;
NETWORK
TITLE = Taktanzahl erreicht ?
//Abfrage ob Taktanzahl erreicht ist
      L     #io_Taktzaehler;
      L     #in_Sollanzahl_Takte;
      >=I;
      S     #io_Taktanzahl_erreicht;
      A     #in_Dauertakt;
      A     #io_Taktanzahl_erreicht;
      JCN   NCCR;	//No Clock Counter Reset
      L     0;
      T     #io_Taktzaehler;
      SET;
      R     #io_Taktanzahl_erreicht;
NCCR: NOP   0;	//No Clock Counter Reset
NETWORK
TITLE = Impuls-Phase des Taktes
//Erhöhung des Zeitzählers während der Impulsphase
//Ist die Sollzeit erreicht wird der Taktzähler erhöht, der Taktausgang 
//zurückgesetzt und der Zeitzähler wieder auf 0 gesetzt
      AN    #io_Taktausgang;
      JC    P_PH;	// wenn Taktausgang nicht gesetzt ist -> Pausephase 
      A     #in_Rueckmeldung;	// solange keine Rückmeldung -> Zeit läuft nicht
      JC    RM_I;
      L     0.000000e+00;
      T     #io_Zeitzaehler;	// Zeitzähler löschen wenn keine Rückmeldung
      JU    ENDE;
RM_I: NOP   0;
      AN    #in_Impuls;
      JC    IMP0;
      L     #in_Impulszeit_in_100ms;
      ITD;
      DTR;
      L     1.000000e-01;
      *R;
      L     #io_Zeitzaehler;	// Zeitzähler erhöhen
      +R;
      T     #io_Zeitzaehler;
      L     #in_Impulszeit;
      <R;
      JC    IMP0;
      SET;
      R     #io_Taktausgang;
      L     #io_Taktzaehler;
      INC   1;
      T     #io_Taktzaehler;
      L     0.000000e+00;
      T     #io_Zeitzaehler;	// Zeitzähler löschen
IMP0: NOP   0;
NETWORK
TITLE = Pause-Phase des Taktes
//Erhöhung des Zeitzählers während der Pausephase
//Ist die Sollzeit erreicht wird der Taktzähler erhöht, der Taktausgang 
//gesetzt und der Zeitzähler wieder auf 0 gesetzt.
//Ist die Solltaktzahl erreicht erfolgt keine weiter Bearbeitung des Netzwerks
P_PH: O     #io_Taktausgang;
      O     #io_Taktanzahl_erreicht;
      JC    ENDE;	// wenn Taktausgang gesetzt ist -> ENDE
      AN    #in_Rueckmeldung;	// solange Rückmeldung -> Zeit läuft nicht
      JC    RM_P;
      L     0.000000e+00;
      T     #io_Zeitzaehler;	// Zeitzähler löschen wenn keine Rückmeldung
      JU    ENDE;
RM_P: NOP   0;
      AN    #in_Impuls;
      JC    ENDE;
      L     #in_Impulszeit_in_100ms;
      ITD;
      DTR;
      L     1.000000e-01;
      *R;
      L     #io_Zeitzaehler;	// Zeitzähler erhöhen
      +R;
      T     #io_Zeitzaehler;
      L     #in_Pausezeit;
      <R;
      JC    ENDE;
      SET;
      S     #io_Taktausgang;
      L     0.000000e+00;
      T     #io_Zeitzaehler;	// Zeitzähler löschen
ENDE: NOP   0;
END_FUNCTION

FUNCTION "FC3 Cycle generator" : VOID	// FC 3
TITLE = Ein- / Ausschaltverzögerung
//Erstellung:
//Datum        Bearbeiter                                                 Version
//--------------------------------------------------------------------------------
//27.05.97     R.Schaffert (sra)                                          01.00.00
//  
//Änderungen:
//Nr. Datum    Bearb Änderung                                       Marke  Version
//--------------------------------------------------------------------------------
//01  05.02.1999  hus      Parameter "Reset" eingeführt             ()    01.01.00
//02  22.03.1999  sra      Fehlerbeseitigung                        ()    01.01.01
//03  25.08.1999  jm       SV inkl. Reset (getestet)                ()    01.02.00
//04  27.09.1999  jm       SI inkl. Reset (getestet)                ()    01.03.00
//05  26.05.2002  jm       SZ inkl. Reset (getestet): Zeitzähler    ()    01.04.00
//06  22.05.2007  sra      Zeitzaehler läuft bei SE weiter          (006) 01.04.01
//
//________________________________________________________________________________
//Beschreibung:
//
//Diese Funktion generiert eine Ein- bzw. Ausschaltverzögerung ohne Verwendung 
//eines Timers. 
//
//Es muß ein Impulssignal "in_Impuls" der Standardimpulse MB4 angelegt werden, 
//das durch die Angabe der Taktzeit in 1/100ms "in_Impulszeit_in_100ms" 
//spezifiziert wird.
//
//Wird der Eingang "Reset" gesetzt, wird der Ausgang zurückgesetzt und der 
//Zeitzähler wird auf 0 gesetzt.
//
//SE: Durch Auswahl von "E" als Verzögerungsart wird eine Einschaltverzögerung 
//gestartet sobald "in_Freigabe" vorhanden ist. Der Ausgang "io_Ausgangssignal" 
//wird nach Ablauf der Verzögerungszeit "in_Verzoegerungszeit" auf 1 gesetzt und 
//steht dann solange an bis die Freigabe nicht mehr vorhanden ist. Der Eingang 
//"in_Reset"  bewirkt eine Nullung der Istzeit und ein Rücksetzen des Ausgangs. 
//Wird der Eingang "in_Reset" weggenommen so startet die Verzögerungszeit von 
//vorne, es sei denn "in_Freigabe" ist dann nicht mehr vorhanden.
//
//SA: Durch Auswahl von "A" als Verzögerungsart wird eine Ausschaltverzögerung 
//gestartet sobald "in_Freigabe" vorhanden ist. Der Ausgang wird sofort mit 
//dem Signal "in_Freigabe" auf 1 gesetzt. Sobald die Freigabe nicht mehr 
//vorhanden ist wird die Ausschaltverzögerung gestartet. Der Ausgang 
//"io_Ausgangssignal" steht weiterhin auf 1. Nach Ablauf der Verzögerungszeit 
//"in_Verzoegerungszeit" wird der Ausgang "io_Ausgangssignal" auf 0 gesetzt. Der 
//Eingang "in_Reset" bewirkt eine Nullung der Istzeit und ein Rücksetzen des 
//Ausgangs. Wird der Eingang "in_Reset" weggenommen so startet die Funktion von 
//vorne, es sei denn "in_Freigabe" ist dann nicht mehr vorhanden.
//
//SV: Durch Auswahl von "V" als Verzögerungsart wird ein verlängerter Impuls 
//gestartet sobald "in_Freigabe" vorhanden ist. Der Ausgang "io_Ausgangssignal" 
//wird für die Verzögerungszeit "in_Verzoegerungszeit" auf 1 gesetzt, unabhängig 
//vom Eingang "in_Freigabe". Der Eingang "in_Reset" bewirkt eine Nullung der 
//Istzeit und ein Rücksetzen des Ausgangs. Wird der Eingang "in_Reset" 
//weggenommen so startet der Impuls von vorne, es sei denn "in_Freigabe" ist dann 
//nicht mehr vorhanden.  
//
//SI: Durch Auswahl von "I" als Verzögerungsart wird ein Impuls gestartet sobald 
//"in_Freigabe" vorhanden ist. Der Ausgang "io_Ausgangssignal" wird für die 
//bestimmte Zeit auf 1 gesetzt, abhängig vom Eingang "in_Freigabe". Der Eingang 
//"Reset" bewirkt eine Nullung der Istzeit und ein Rücksetzen des Ausgangs 
//"io_Ausgangssignal". Wird der Eingang "Reset" weggenommen so startet der Impuls 
//von vorne, es sei denn "in_Freigabe" ist dann nicht mehr vorhanden.
//
//SZ: Diese Funktion kann als Zeitzähler bezeichnet werden. Sobald "in_Freigabe" 
//vorhanden ist wird die Zeit hochgezählt. Ohne "in_Freigabe" bleibt die Zeit 
//stehen, sobald "in_Freigabe" wieder vorhanden ist wird weiter gezählt. Ist die 
//Sollzeit "in_Verzoegerungszeit" erreicht und "in_Freigabe" geht weg, wird der 
//Zeitzähler rückgesetzt. Der Eingang "Reset" bewirkt eine Nullung der Istzeit 
//und ein Rücksetzen des Ausgangs "io_Ausgangssignal". Wird der Eingang "Reset" 
//weggenommen so startet der Zeitzähler von vorne, es sei denn "in_Freigabe" ist 
//dann nicht mehr vorhanden.
AUTHOR : hus
FAMILY : AZO
VERSION : 0.1
VAR_INPUT
  in_Freigabe : BOOL ;	//Freigabe Timernachbildung
  in_Reset : BOOL ;	//Reset (z.B. Steuerspannung aus)
  in_Impuls : BOOL ;	//Impulseingang (M1.7)
  in_Impulszeit_in_100ms : INT ;	//Impulszeit in 100ms (MW6)
  in_Verzoegerungsart : CHAR ;	//'E'=Einschalt-,'A'=Ausschaltverz.,'V'=verl.Impuls,'I'= Impuls,'Z'=Zeitzähler
  in_Verzoegerungszeit : REAL ;	//Verzögerungszeit in Sekunden
END_VAR
VAR_IN_OUT
  io_Ausgangssignal : BOOL ;	//Timerausgang
  io_Zeitzaehler : REAL ;	//Zeitzähler (abgelaufene Zeit)
END_VAR
BEGIN
NETWORK
TITLE = Einschaltverzögerung
//Einschaltverzögerung
      L     #in_Verzoegerungsart;
      L     'E';
      <>I;
      JC    E1;
      A     #in_Freigabe;
      JC    SE;
      SET;
      R     #io_Ausgangssignal;
      L     0.000000e+00;
      T     #io_Zeitzaehler;
      JU    E1;
//    O     #io_Ausgangssignal // (006)
SE:   ON    #in_Impuls;
      JC    E1;
      L     #in_Impulszeit_in_100ms;
      ITD;
      DTR;
      L     1.000000e-01;
      *R;
      L     #io_Zeitzaehler;
      +R;
      T     #io_Zeitzaehler;
      L     #in_Verzoegerungszeit;
      >=R;
      S     #io_Ausgangssignal;
E1:   NOP   0;
NETWORK
TITLE = Ausschaltverzögerung
//Ausschaltverzögerung
      L     #in_Verzoegerungsart;
      L     'A';
      <>I;
      JC    E2;
      AN    #in_Freigabe;
      JC    SA;
      SET;
      S     #io_Ausgangssignal;
      L     0.000000e+00;
      T     #io_Zeitzaehler;
      JU    E2;
SA:   ON    #io_Ausgangssignal;
      ON    #in_Impuls;
      JC    E2;
      L     #in_Impulszeit_in_100ms;
      ITD;
      DTR;
      L     1.000000e-01;
      *R;
      L     #io_Zeitzaehler;
      +R;
      T     #io_Zeitzaehler;
      L     #in_Verzoegerungszeit;
      >=R;
      R     #io_Ausgangssignal;
E2:   NOP   0;
NETWORK
TITLE = Verlängerter Impuls
//Verlängerter Impuls
      L     #in_Verzoegerungsart;
      L     'V';
      <>I;
      JC    E3;
      O     #in_Freigabe;
      O     #io_Ausgangssignal;
      JC    SV;
      CLR;
      =     #io_Ausgangssignal;
      L     0.000000e+00;
      T     #io_Zeitzaehler;
      JU    E3;
SV:   A     #in_Freigabe;
      S     #io_Ausgangssignal;
      L     #io_Zeitzaehler;
      L     #in_Verzoegerungszeit;
      >=R;
      R     #io_Ausgangssignal;
      ON    #in_Impuls;
      ON    #io_Ausgangssignal;
      JC    E3;
      L     #in_Impulszeit_in_100ms;
      ITD;
      DTR;
      L     1.000000e-01;
      *R;
      L     #io_Zeitzaehler;
      +R;
      T     #io_Zeitzaehler;
      L     #in_Verzoegerungszeit;
      >=R;
      R     #io_Ausgangssignal;
E3:   NOP   0;
NETWORK
TITLE = Impuls
//Impuls
      L     #in_Verzoegerungsart;
      L     'I';
      <>I;
      JC    E4;
      A     #in_Freigabe;
      JC    SI;
      CLR;
      =     #io_Ausgangssignal;
      L     0.000000e+00;
      T     #io_Zeitzaehler;
      JU    E4;
SI:   A     #in_Freigabe;
      S     #io_Ausgangssignal;
      L     #io_Zeitzaehler;
      L     #in_Verzoegerungszeit;
      >=R;
      R     #io_Ausgangssignal;
      ON    #in_Impuls;
      ON    #io_Ausgangssignal;
      JC    E4;
      L     #in_Impulszeit_in_100ms;
      ITD;
      DTR;
      L     1.000000e-01;
      *R;
      L     #io_Zeitzaehler;
      +R;
      T     #io_Zeitzaehler;
      L     #in_Verzoegerungszeit;
      >=R;
      R     #io_Ausgangssignal;
E4:   NOP   0;
NETWORK
TITLE = Zeitzähler 'Z'
//Einschaltverzögerung
      L     #in_Verzoegerungsart;
      L     'Z';
      <>I;
      JC    E5;
      AN    #in_Freigabe;
      A     #io_Ausgangssignal;
      JCN   SZ;	// Zeitzähler wird gelöscht, wenn Zeit abgelaufen und FRG weg geht
      SET;
      R     #io_Ausgangssignal;
      L     0.000000e+00;
      T     #io_Zeitzaehler;
      JU    E5;
SZ:   O     #io_Ausgangssignal;
      ON    #in_Freigabe;
      ON    #in_Impuls;
      JC    E5;
      L     #in_Impulszeit_in_100ms;
      ITD;
      DTR;
      L     1.000000e-01;
      *R;
      L     #io_Zeitzaehler;
      +R;
      T     #io_Zeitzaehler;
      L     #in_Verzoegerungszeit;
      >=R;
      S     #io_Ausgangssignal;
E5:   NOP   0;
NETWORK
TITLE = Rücksetzen Ausschaltverzögerung wenn Reseteingang = "True". 
      AN    #in_Reset;
      JC    E6;
      A     #io_Ausgangssignal;
      R     #io_Ausgangssignal;
      L     0.000000e+00;
      T     #io_Zeitzaehler;
E6:   NOP   0;
END_FUNCTION

FUNCTION "FC5 Block Transfer" : VOID	// FC 5
TITLE = BlockTransfer
//Erstellung:
//Datum        Bearbeiter                                                 Version
//--------------------------------------------------------------------------------
//26.06.97     G.Herkert (hkt)                                            01.00.00
//
//Änderungen:
//Nr. Datum    Bearb Beschreibung                                   Marke Version
//--------------------------------------------------------------------------------
//01  20.05.98 sra   komplette Überarbeitung                              02.00.00
//02  29.10.98 gea   Überprüfung Länge und Existenz DBs                   02.01.00
//03  24.11.98 gea   'I' kopiert in/von akt Instanz-DB                    02.02.00
//04  10.05.99 sra   Bereichszeigerberechnung korrigiert                  02.02.01
//05  10.12.01 gea   'K' löscht Bereich                             (005) 02.03.00
//06  07.06.10 sra   Bereich > 32767 kopieren                       (006) 02.03.01
//
//________________________________________________________________________________
//Funktion:
//
//Blocktranferfunktion mit Systemfunktion SFC20
//-Bei "Quell_Typ" = 'E' werden die Aktualwerte der in "Quell_DW" definierten 
// Eingangsadressen ausgelesen und kopiert.
//-Bei "Quell_Typ" = 'A' werden die Aktualwerte der in "Quell_DW" definierten 
// Ausgangsadressen ausgelesen und kopiert.
//-Bei "Quell_Typ" = 'M' werden die Aktualwerte der in "Quell_DW" definierten 
// Merkeradressen ausgelesen und kopiert.
//-Bei "Quell_Typ" = 'D' werden die Aktualwerte der in "Quell-DB" und "Quell_DW"  
// definierten Datenworte ausgelesen und kopiert.
//-Bei "Quell_Typ" = 'I' werden die Aktualwerte der in "Quell_DW" definierten 
// Datenworte des aktuellen Instanz-DBs ausgelesen und kopiert.
//
//-Bei "Ziel_Typ" = 'E' werden die definierten Quelldaten an den durch 
// "in_Ziel_DW" definierten Eingangsbereich kopiert.
//-Bei "Ziel_Typ" = 'A' werden die definierten Quelldaten an den durch 
// "in_Ziel_DW" definierten Ausgangsbereich kopiert.
//-Bei "Ziel_Typ" = 'M' werden die definierten Quelldaten an den durch 
// "in_Ziel_DW" definierten Merkerbereich kopiert.
//-Bei "Ziel_Typ" = 'D' werden die definierten Quelldaten an den durch  
//"in_Ziel_DB" und "in_Ziel_DW" definierten Global-Datenbaustein kopiert.
//-Bei "Ziel_Typ" = 'I' werden die definierten Quelldaten an den durch  
// "in_Ziel_DW" definierten Zielbereich des aktuellen Instanz-Datenbausteines  
// kopiert.
//
//An den SFC20 werden Zeiger (ANY-Zeiger) angelegt die die Quelle und das Ziel 
//beschreiben. Zeiger sind folgendermaßen aufgebaut:
//     Byte n       B#16#10 
//     Byte n+1     Datentyp (Bool, Byte, usw.)
//     Byte n+2     Anzahl der Datentypen die kopiert werdn sollen (2 Byte)
//     Byte n+4     Datenbausteinnummer (2 Byte)
//     Byte n+6     Bereichszeiger (4 Byte)
//
//Aufbau des bereichsübergreifenden Zeigers:  10000ZZZ 00000yyy yyyyyyyy yyyyyxxx
//      z = Operandenbereich (codiert)
//      y = Byte-Adresse
//      x = Bit-Adresse
AUTHOR : hkt
FAMILY : AZO
VERSION : 0.0
VAR_INPUT
  Quell_Typ : CHAR ;	//E=Eingang, A=Ausgang, M=Merker, D=DB, I=Instanz-DB, K=Löschen
  Quell_DB : INT ;	//Quell-Datenbaustein bei DW-Transfer
  Quell_DW : INT ;	//Quell-Datenwort, Byte-Adresse der Quelle
  Ziel_Typ : CHAR ;	//E=Eingang, A=Ausgang, M=Merker, D=DB, I=Instanz-DB
  Ziel_DB : INT ;	//Ziel-Datenbaustein bei DW-Transfer
  Ziel_DW : INT ;	//Ziel-Datenwort, Byte-Adresse des Zieles
  Block_Laenge : INT ;	//Blocklänge in Byte
END_VAR
VAR_OUTPUT
  outFehler : INT ;	//1=Ziel-Typ ungültig, 2=DB existiert nicht, 3= DB zu kurz, SFC20 Fehlermeldung
END_VAR
VAR_TEMP
  Quellzeiger : ANY ;
  Zielzeiger : ANY ;
  SFC20_return : INT ;
  Operandenbereich : INT ;
  DB_Test_Nr : WORD ;
  DB_Test_Fehler : INT ;
  DB_Test_Anz_Byte : WORD ;
  DB_Test_Schreib_Schutz : BOOL ;
END_VAR
BEGIN
NETWORK
TITLE = Bereich in DB-löschen
//(005)
      A(;
      L     #Quell_Typ;
      L     'K';
      ==I;
      );
      A(;
      L     #Ziel_Typ;
      L     'D';
      ==I;
      );
      JCN   BLOE;
      CALL  "FC30 Pre -assign DB" (
           DB_Nr                    := #Ziel_DB,
           DW_Anfang                := #Ziel_DW,
           Anzahl_Bytes             := #Block_Laenge,
           Wert                     := 0);
      BEU;
BLOE: NOP   0;
NETWORK
TITLE = Operandenbereich Quelle codieren
//Bereichscodierung für Quelltyp durchführen
//Operandenbereich im bereichsübergreifenden Zeiger
//
//Aufbau des bereichsübergreifenden Zeigers:  10000ZZZ 00000yyy yyyyyyyy yyyyyxxx
//      z = Operandenbereich (codiert)
//      y = Byte-Adresse
//      x = Bit-Adresse
//    
      L     #Quell_Typ;
      L     'E';	// Quelle = Eingänge
      ==I;
      L     1;
      JC    M001;
      L     #Quell_Typ;
      L     'A';	// Quelle = Ausgänge
      ==I;
      L     2;
      JC    M001;
      L     #Quell_Typ;
      L     'M';	// Quelle = Merker
      ==I;
      L     3;
      JC    M001;
      L     #Quell_Typ;
      L     'D';	// Quelle = DB (Globaldaten)
      ==I;
      L     4;
      JC    M001;
      L     #Quell_Typ;
      L     'I';	// Quelle = Instanz-DB
      ==I;
      L     5;
      JC    M001;
      L     #Quell_Typ;
      L     'L';	// Quelle = Temporäre-Lokal-Daten
      ==I;
      L     6;
      JC    M001;
      L     #Quell_Typ;
      L     'V';	// Quelle = temp. Lokaldaten des Vorgängerbausteins
      ==I;
      L     7;
      JC    M001;
      L     1;	// Kein gültiger Parameter -> Fehler und Ende
      T     #outFehler;
      BEU;
M001: T     #Operandenbereich;
NETWORK
TITLE = Quell-Datenbaustein prüfen
//Überprüfen bei Quelltyp = D,I : Baustein existiert und ist ausreichend lang
      L     #Operandenbereich;
      L     5;	//Quelle ist Instanz-DB 
      <>I;
      JC    M004;
      L     DINO;	//Nummer akt. Instanz-DB
      T     #Quell_DB;
      T     #DB_Test_Nr;
      JU    M005;
M004: L     #Operandenbereich;
      L     4;	//Quelle ist Global-DB
      <>I;
      JC    M003;
      L     #Quell_DB;
      T     #DB_Test_Nr;
M005: CALL  "SFC 24 TEST_DB" (
           DB_NUMBER                := #DB_Test_Nr,
           RET_VAL                  := #DB_Test_Fehler,
           DB_LENGTH                := #DB_Test_Anz_Byte,
           WRITE_PROT               := #DB_Test_Schreib_Schutz);
      L     #DB_Test_Fehler;
      L     0;
      ==I;
      JC    M006;
      L     2;	//DB existiert nicht
      T     #outFehler;
      BEU;
M006: L     #Quell_DW;
      L     #Block_Laenge;
      +D;	// (006)    
      L     #DB_Test_Anz_Byte;
      <=D;	// (006)    
      JC    M003;
      L     3;	//DB nicht ausreichend lang
      T     #outFehler;
      BEU;
M003: NOP   0;
NETWORK
TITLE = Quellezeiger belegen
//Quelle vom Typ "ANY" erstellen
      LAR1  P##Quellzeiger;
      L     B#16#10;
      T     LB [AR1,P#0.0];	//Syntax-ID ist immer 10h bei AWL
      L     2;
      T     LB [AR1,P#1.0];	// Datentyp = 2 (Byte)
      L     #Block_Laenge;
      T     LW [AR1,P#2.0];	// Anzahl der Bytes die kopiert werden sollen
      L     #Quell_DB;
      T     LW [AR1,P#4.0];	// Datenbaustzeinnummer
      L     #Operandenbereich;
      L     128;	// 128 addieren (Bit 31 muß 1 sein)
      +I;
      SLD   24;	// 24 Stellen nach rechts schieben
      L     #Quell_DW;
      SLD   3;	// Quell-DW an Byte-Adresse schieben 
      +D;	// Zeiger zusammenfügen
      T     LD [AR1,P#6.0];	// siehe Aufbau Bereichszeiger NW1
NETWORK
TITLE = Operandenbereich Ziel codieren
//Bereichscodierung für Zieltyp durchführen
//Operandenbereich im bereichsübergreifenden Zeiger
//
//Aufbau des bereichsübergreifenden Zeigers:  10000ZZZ 00000yyy yyyyyyyy yyyyyxxx
//      z = Operandenbereich (codiert)
//      y = Byte-Adresse
//      x = Bit-Adresse
//    
      L     #Ziel_Typ;
      L     'E';	// Ziel = Eingänge
      ==I;
      L     1;
      JC    M002;
      L     #Ziel_Typ;
      L     'A';	// Ziel = Ausgänge
      ==I;
      L     2;
      JC    M002;
      L     #Ziel_Typ;
      L     'M';	// Ziel = Merker
      ==I;
      L     3;
      JC    M002;
      L     #Ziel_Typ;
      L     'D';	// Ziel = DB (Globaldaten)
      ==I;
      L     4;
      JC    M002;
      L     #Ziel_Typ;
      L     'I';	// Ziel = Instanz-DB
      ==I;
      L     5;
      JC    M002;
      L     #Ziel_Typ;
      L     'L';	// Ziel = Temporäre-Lokal-Daten
      ==I;
      L     6;
      JC    M002;
      L     #Ziel_Typ;
      L     'V';	// Ziel = temp. Lokaldaten des Vorgängerbausteins
      ==I;
      L     7;
      JC    M002;
      L     1;	// Kein gültiger Parameter -> Fehler und Ende
      T     #outFehler;
      BEU;
M002: T     #Operandenbereich;
NETWORK
TITLE = Ziel-Datenbaustein prüfen
//Überprüfen bei Zieltyp = D,I : Baustein existiert und ist ausreichend lang
      L     #Operandenbereich;
      L     5;	//Ziel ist Instanz-DB 
      <>I;
      JC    M007;
      L     DINO;	//Nummer akt. Instanz-DB
      T     #Ziel_DB;
      T     #DB_Test_Nr;
      JU    M008;
M007: L     #Operandenbereich;
      L     4;	//Ziel ist Global-DB
      <>I;
      JC    M010;
      L     #Ziel_DB;
      T     #DB_Test_Nr;
M008: CALL  "SFC 24 TEST_DB" (
           DB_NUMBER                := #DB_Test_Nr,
           RET_VAL                  := #DB_Test_Fehler,
           DB_LENGTH                := #DB_Test_Anz_Byte,
           WRITE_PROT               := #DB_Test_Schreib_Schutz);
      L     #DB_Test_Fehler;
      L     0;
      ==I;
      JC    M009;
      L     2;	//DB existiert nicht
      T     #outFehler;
      BEU;
M009: L     #Ziel_DW;
      L     #Block_Laenge;
      +D;	// (006)    
      L     #DB_Test_Anz_Byte;
      <=D;	// (006)    
      JC    M010;
      L     3;	//DB nicht ausreichend lang
      T     #outFehler;
      BEU;
M010: NOP   0;
NETWORK
TITLE = Zielzeiger belegen
//Ziel vom Typ "ANY" erstellen
      LAR1  P##Zielzeiger;
      L     B#16#10;
      T     LB [AR1,P#0.0];	//Syntax-ID ist immer 10h bei AWL
      L     2;
      T     LB [AR1,P#1.0];	// Datentyp = 2 (Byte)
      L     #Block_Laenge;
      T     LW [AR1,P#2.0];	// Anzahl der Bytes die kopiert werden sollen
      L     #Ziel_DB;
      T     LW [AR1,P#4.0];	// Datenbaustzeinnummer
      L     #Operandenbereich;
      L     128;	// 128 addieren (Bit 31 muß 1 sein)
      +I;
      SLD   24;	// 24 Stellen nach rechts schieben
      L     #Ziel_DW;
      SLD   3;	// Quell-DW an Byte-Adresse schieben 
      +D;	// Zeiger zusammenfügen
      T     LD [AR1,P#6.0];	// siehe Aufbau Bereichszeiger NW1
NETWORK
TITLE = Blocktransfer
//Blocktransfer mit Systemfunktion SFC20
      CALL  "SFC 20 BLKMOV" (
           SRCBLK                   := #Quellzeiger,
           RET_VAL                  := #SFC20_return,
           DSTBLK                   := #Zielzeiger);
NETWORK
TITLE = Rückgabewert SFC20
//Rückgabewert des SFC20 übergeben
      L     #SFC20_return;
      T     #outFehler;
END_FUNCTION

FUNCTION "FC7 Read Table" : VOID	// FC 7
TITLE = Tabelle auslesen
//Erstellung:
//Datum        Bearbeiter                                                 Version
//--------------------------------------------------------------------------------
//30.10.98     A.Geiger (gea)                                             01.00.00
//
//Änderungen:
//Nr. Datum    Bearb Beschreibung                                   Marke Version
//--------------------------------------------------------------------------------
//01  10.05.99 sra   Bereichszeigerberechnung korrigiert                  01.00.01
//02  29.08.00 gea   Neue Konzeption(Kopieren über Schleife)              02.00.00
//03  26.10.01 gea   Fehlerbehebung DB überprüfen                   (003) 02.00.01
//04  26.10.01 gea   Fehler bei Anfangsbyte negativ                 (004) 02.00.02
//05  29.02.16 sra   Anpassung für Tabellen > 32767 Byte            (005) 02.00.03
//06  17.06.16 sra   Fehlerbeseitigung Zeigerberechnung             
//                   negative Zeilen sind ebenfalls möglich         (006) 02.00.04
//________________________________________________________________________________
//Funktion:
//
//Beschreibung: Datensatz aus Tabelle auslesen
//
//Aufbau Tabellen-DB:
//      DBB(Offset)    ... DBB(n-1)  1.Zeile
//      DBB(Offset+n)  ... DBB(2n-1) 2.Zeile
//      DBB(Offset+2n) ... DBB(3n-1) 3.Zeile
//      usw.
//
//Die Anzahl der Spalten pro Zeile (n) ist abhängig von der Länge des "Ziels".
//Das "Ziel" muß ein ANY-Zeiger auf Bytes oder eine Stuktur sein.
//Eine Überprüfung auf Existenz und Länge des Tabellen-DBs wird durchgeführt.
//
//Fehlermeldungen:
//-1 = Bereichszeiger Quelle falsch
//-2 = Bereichszeiger Ziel falsch
//-3 = Blocklänge falsch
//-4 = Datenbaustein nicht existent 
//-5 = Datenbaustein Längenfehler
//-6 = Fehler Datentyp in ANY-Zeiger
//-7 = Fehler Anfangsbyte negativ    
//
AUTHOR : gea
FAMILY : gea
VERSION : 0.0
VAR_INPUT
  in_Tabelle_DB : INT ;	//Tabellen-DB-Nr.
  in_Offset_DW : INT ;	//Offset erster Tabelleneintrag in Tabellen-DB
  in_Zeile_lesen : INT ;	//Eintrag in Tabelle, der gelesen werden soll
END_VAR
VAR_OUTPUT
  out_Fehler : INT ;	//-1=Q,-2=Z,-3=Blocklänge,-4=DB n. vorh.,-5=DB zu kurz,-6=Datentyp,-7=Anfangsbyte
END_VAR
VAR_IN_OUT
  io_Ziel : ANY ;	//Zeiger auf Zieldaten Block in den kopiert wird
END_VAR
VAR_TEMP
  G_DB_SAVE : INT ;	//Global-DB-Register
  I_DB_SAVE : INT ;	//Instanz-DB-Register
  Zeiger_Quelle : DWORD ;
  DB_Quelle : INT ;
  Zeiger_Ziel : DWORD ;
  DB_Ziel : INT ;
  Blocklaenge : INT ;
  Datentyp : BYTE ;
  Start_DBB : INT ;
END_VAR
BEGIN
NETWORK
TITLE = DB-Register sichern
      L     DBNO;
      T     #G_DB_SAVE;
      L     DINO;
      T     #I_DB_SAVE;
NETWORK
TITLE = ANY-Zeiger Ziel zerlegen
      L     P##io_Ziel;
      LAR1;
      L     B [AR1,P#1.0];
      T     #Datentyp;
      L     W [AR1,P#2.0];
      T     #Blocklaenge;
      L     W [AR1,P#4.0];
      T     #DB_Ziel;
      L     D [AR1,P#6.0];
      L     DW#16#FFFFFF;	// (006)
      AD;	// (006)
      T     #Zeiger_Ziel;
NETWORK
TITLE = Blocklänge prüfen
      L     #Blocklaenge;
      L     0;
      <=I;
      JC    BLFE;	//Blocklänge Fehler
NETWORK
TITLE = Datentyp prüfen
      L     #Datentyp;
      L     2;	//Datentyp = Byte oder Struct
      ==I;
      JCN   DTFE;
NETWORK
TITLE = Start-DBB des gewählten Eintrags
      L     #in_Zeile_lesen;
      L     1;
      -I;
      L     #Blocklaenge;
      *I;
      L     #in_Offset_DW;
      +I;
      T     #Start_DBB;	//Start des n-ten Eintrags
//      L     #Start_DBB                  //Start des n-ten Eintrags      //(004) // (006)
//      L     0                           //                                (004) // (006)
//      >=I                               //                                (004) // (006)
//      SPBN  DBBN                        //Fehler Anfangsbyte negativ    //(004) // (006)
NETWORK
TITLE = Bereichszeiger Quellzeiger
      L     W#16#84;
      CAD;
      L     #Start_DBB;
      SLD   3;
      +D;
      T     #Zeiger_Quelle;
NETWORK
TITLE = Quell-DB
      L     #in_Tabelle_DB;
      T     #DB_Quelle;
NETWORK
TITLE = DBs aufschlagen
//      L     #DB_Quelle                               //(003)
//      L     0                                        //(003)
//      <>I                                            //(003)
//      SPBN  QNDB                                     //(003)
      OPN   DB [#DB_Quelle];
      L     DBNO;
      L     0;
      <=I;
      JC    DBNX;	//Fehler DB existiert nicht
      L     #Start_DBB;
      L     #Blocklaenge;
      +D;	// (005)
      L     DBLG;
      >D;	// (005)
      JC    DBLF;	//Fehler DB Länge nicht ausreichend
      L     #DB_Ziel;
      L     0;
      <>I;
      JCN   ZNDB;
      OPN   DI [#DB_Ziel];
      L     DINO;
      L     0;
      <=I;
      JC    DBNX;	//Fehler DB existiert nicht
      L     #Zeiger_Ziel;
      SRD   3;	//Anfangsbyte (005)
      L     #Blocklaenge;
      +D;	// (005)
      L     DILG;
      >D;	// (005)
      JC    DBLF;	//Fehler DB Länge nicht ausreichend
      L     #Zeiger_Ziel;
      L     DW#16#FFFFFF;
      AD;
      L     W#16#85;
      CAD;
      +D;
      T     #Zeiger_Ziel;
ZNDB: NOP   0;
NETWORK
TITLE = Bytes kopieren
//geschwindigkeitsopitmiert:
//- Schleifenzäehler bleibt in AKKU1 und AKKU2
//- Kopieren über Worte, letztes Byte (ungerade Bytezahl) separat.
// (network holds code this reader does not know; not shown)
NETWORK
TITLE = Fehlerauswertung
      L     0;	//kein Fehler
      JU    SEFE;	//  setze Fehlerausgang
      L     -1;	//Bereichszeiger Quelle falsch
      JU    SEFE;	//  setze Fehlerausgang
      L     -2;	//Bereichszeiger Ziel falsch
      JU    SEFE;	//  setze Fehlerausgang
BLFE: L     -3;	//Blocklänge falsch
      JU    SEFE;	//  setze Fehlerausgang
DBNX: L     -4;	//Datenbaustein nicht existent 
      JU    SEFE;	//  setze Fehlerausgang
DBLF: L     -5;	//Datenbaustein Längenfehler
      JU    SEFE;	//  setze Fehlerausgang
DTFE: L     -6;	//Fehler Datentyp in ANY-Zeiger
      JU    SEFE;	//  setze Fehlerausgang         (004)
      L     -7;	//Fehler Anfangsbyte negativ    (004)
SEFE: T     #out_Fehler;
NETWORK
TITLE = DB-Register wiederherstellen
      OPN   DB [#G_DB_SAVE];
      OPN   DI [#I_DB_SAVE];
NETWORK
TITLE = BIE-Bit zuweisen
      L     #out_Fehler;
      L     0;
      ==I;
      SAVE;
END_FUNCTION

FUNCTION "FC10 Analogue value r/w" : VOID	// FC 10
TITLE = Analogwert lesen/schreiben
//Erstellung:
//Datum        Bearbeiter                                                 Version
//--------------------------------------------------------------------------------
//06.08.97     G.Herkert (hkt)                                            01.00.00
//
//Änderungen:
//Nr. Datum    Bearb Beschreibung                                   Marke Version
//--------------------------------------------------------------------------------
//01  21.10.97 rh    Drahtbruchüberwachung ergänzt                        01.01.00
//02  05.12.97 rh    Adressen auf PEW und PAW geändert                    01.01.01
//03  25.11.98 gea   Simulation eingefügt                                 01.02.00
//04  29.03.99 gea   Fehlerbehebung Drahtbruchüberwachung                 01.02.01
//05  30.06.99 sra   Fehlerbehebung Drahtbruchüberwachung                 01.02.02
//06  19.02.00 sra   Unterscheidung Drahtbruchüberwachung                 01.02.03
//07  12.09.01 gea   Eingangsparameter in_E_A_Adresse als INT             01.03.00
//08  16.03.04 sra   nicht in Simulations-DB schreiben wenn Simul aus     01.03.01
//09  17.09.08 sra   Wago-System 750-466 erweitert                  (009) 01.04.00
//________________________________________________________________________________
//Funktion:
//
//Der Baustein liest den Wert eines Analogeinganges ein und normiert diesen. Die 
//Normierung erfolgt anhand der Vorgabe der Eingangsparameter Obergrenze und 
//Untergrenze.
//
//Hinweis:
//- bei Siemens-Baugruppen ist der Wert "MaxDigit" = 27648
//- bei Wago-Baugruppen 740-466 ist der Wert "MaxDigit" = 32760
//
//
AUTHOR : hkt
FAMILY : AZO
VERSION : 0.0
VAR_INPUT
  in_E_A : CHAR  := 'E';	//E = Eingang, A = Ausgang
  in_EA_Adresse : INT ;	//Ein-/Ausgangsadresse des Analogkanals
  in_OberGrenze : REAL ;	//Obergrenze des Ausgabewertes (z.B. Drucktransmitter: 2 bar)
  in_UnterGrenze : REAL ;	//Untergrenze des Ausgabewertes (z.B. Drucktransmitter: 0 bar)
  in_MaxDigit : REAL ;	//Digitwert den die Baugruppe bei der Obergrenze liefert z.B. 27648
  in_MinDigit : REAL ;	//Digitwert den die Baugruppe bei der Untergrenze liefert z.B. 0 bzw. -27648
  in_Typ : CHAR ;	//Z=Zentralbaugruppe, B=ET200B Analogmodul, W=Wago 750-466, sonstige
  in_Simulation : BOOL ;	//Simulation des Analogwertes über Eintrag in Datenbaustein
  in_DB_Simulation_EA : INT ;	//Simulation-DB des Analogwertes über Eintrag in Datenbaustein
END_VAR
VAR_IN_OUT
  io_Wert : REAL ;	//eingelesener und normierter Wert den die Baugrppe liefert
  io_Drahtbruch : BOOL ;	//Drahtbruchstoerung
END_VAR
VAR_TEMP
  MaxDigit_MinDigit : REAL ;
  E_MinDigit : REAL ;
  OG_UG : REAL ;
  Eingang_Real : REAL ;
  Pointer_EA_Adresse : DWORD ;
  Wert_analog : WORD ;
  DB_Sim : INT ;
END_VAR
BEGIN
NETWORK
TITLE = Zwischenwerte berechnen
      L     #in_MaxDigit;
      L     #in_MinDigit;
      -R;
      T     #MaxDigit_MinDigit;
      L     #in_OberGrenze;
      L     #in_UnterGrenze;
      -R;
      T     #OG_UG;
NETWORK
TITLE = Zeiger berechnen
// Zeiger auf EA-Adresse berechnen
      LAR1  P#0.0;
      L     #in_EA_Adresse;
      SLW   3;
      +AR1;
      LAR1;
      T     #Pointer_EA_Adresse;	//Zeiger auf EA-Adresse
      L     #in_DB_Simulation_EA;
      T     #DB_Sim;	//Zeiger auf EA-DB
NETWORK
TITLE = Analogwert einlesen
//Analogwert einlesen
//Formel:   Wert = UG + (OG-UG)*(E-MinDigit) / (MaxDigit-MminDigit)
      L     #in_E_A;
      L     'E';
      <>I;
      JC    NotE;
      A     #in_Simulation;
      JC    SIME;
      L     PIW [#Pointer_EA_Adresse];
      JU    WERE;	// (008)
SIME: OPN   DB [#DB_Sim];
      L     DBW [#Pointer_EA_Adresse];
WERE: T     #Wert_analog;
      A(;
      L     #in_Typ;	// Abfrage Drahtbruchüberwachung
      L     'Z';	// "Z" = Zentralbaugruppe
      ==I;
      );
      A(;
      L     #Wert_analog;	// 7FFF Ersatzwert für Drahtbruch
      L     W#16#7FFF;
      ==I;
      );
      O;
      A(;
      L     #in_Typ;	// Abfrage Drahtbruchüberwachung
      L     'B';	// "B" = ET200B Baugruppe
      ==I;
      );
      A(;
      L     #Wert_analog;	// 8000 Ersatzwert für Drahtbruch
      L     W#16#8000;
      ==I;
      );
      O;	// -> (009)
      A(;
      L     #in_Typ;	// Abfrage Kartentyp
      L     'W';	// "W" = Wago System 750-466
      ==I;	// Karte meldet mit den rechten 3 Bis ein Kurzschluss bzw. Überlauf
      );
      A(;
      L     #Wert_analog;
      L     W#16#7;
      AW;
      L     W#16#0;
      <>I;
      );	// <- (009)
      =     #io_Drahtbruch;
      L     #Wert_analog;
      ITD;
      DTR;
      T     #Eingang_Real;
      L     #Eingang_Real;
      L     #in_MinDigit;
      -R;
      T     #E_MinDigit;
      L     #OG_UG;
      L     #E_MinDigit;
      *R;
      L     #MaxDigit_MinDigit;
      /R;
      L     #in_UnterGrenze;
      +R;
      T     #io_Wert;
NotE: NOP   0;
NETWORK
TITLE = AnalogWert ausgeben:  
//AnalogWert ausgeben:
//Formel : A = MinDigit+(MaxDigit-MinDigit)*(Wert-UG)/ (Og-UG)
      L     #in_E_A;
      L     'A';
      <>I;
      JC    NotA;
      L     #io_Wert;
      L     #in_UnterGrenze;
      -R;
      L     #OG_UG;
      /R;
      L     #MaxDigit_MinDigit;
      *R;
      L     #in_MinDigit;
      +R;
      RND;
      T     #Wert_analog;
      A     #in_Simulation;
      JC    SIMA;
      T     PQW [#Pointer_EA_Adresse];
      JU    NotA;	// (008)
SIMA: OPN   DB [#DB_Sim];
      T     DBW [#Pointer_EA_Adresse];
NotA: NOP   0;
END_FUNCTION

FUNCTION "FC11 PressureTransmitter" : VOID	// FC 11
TITLE = Drucktransmitter
//Erstellung:
//Datum        Bearbeiter                                                 Version
//--------------------------------------------------------------------------------
//20.10.1999   M. Junker (jm)                                             01.00.00
//
//
//Änderungen:
//Nr. Datum    Bearb Beschreibung                                   Marke Version
//--------------------------------------------------------------------------------
//01  03.11.99 jm    Druckstörung löschen ohne FRG                        01.00.01
//
//________________________________________________________________________________
//Funktion:
//
//Der Baustein gleicht Abweichungen eines eingelesenen Förderdruckes so ab, daß 
//bei aktuellem Luftdruck der Wert "0" ausgegeben wird. 
//Der Abgleich erfolgt, wenn das Eingangssignal "Gebäse aktiv" für eine gewisse 
//Zeit (Parameter "Verz_Abgleich") nicht mehr ansteht.
//Weiterhin wird der Druckwert überwacht und bei Überschreitung des Max-Druckes 
//eine Störmeldung erzeugt. Das Rücksetzen dieser Störmeldung erfolgt erst, wenn 
//der Min-Druck wieder unterschritten ist.
//
AUTHOR : jm
FAMILY : AZO
VERSION : 0.0
VAR_INPUT
  AbsolutDruck : REAL ;	//eingelesener Analogwert
  MinDruck : REAL ;	//Min. Druck: bei Unterschreitung wird Druckstörung rückgesetzt
  MaxDruck : REAL ;	//Max. Druck: bei Überschreitung erfolgt Störmeldung
  LeerDruck : REAL ;	//Leerdruck: bei Unterschreitung wird Parameter "Leerdruck aktiv" gesetzt
  Verz_Abgleich : REAL ;	//Verzögerung Abgleich
  Auswahl_S_D : CHAR ;	//Auswahl Saug-/Druckförderung
  Drahtbruch : BOOL ;	//Drahtbruchmeldung von Analogkanal
  Geblaese_aktiv : BOOL ;	//Gebläse/Pumpe aktiv
  FRG_Druckstoerung : BOOL ;	//Freigabe Druckstoerung
END_VAR
VAR_IN_OUT
  Zeitzaehler : REAL ;	//Zeitzaehler für Verzögerung Abgleich
  RelativDruck : REAL ;	//Relativdruck
  MemoryDruck : REAL ;	//Memory-Feld für Abgleich
  Druckstoerung : BOOL ;	//Ausgabe Druckstoerung
  Leerdruck_aktiv : BOOL ;	//Leerdruck unterschritten
  Ausgang_Timer : BOOL ;	//Ausgangssignal Timernachbildung Verzögerung Abgleich
END_VAR
BEGIN
NETWORK
TITLE = Verzögerung Druckabgleich
      CALL  "FC3 Cycle generator" (
           in_Freigabe              := #Geblaese_aktiv,
           in_Reset                 := FALSE,
           in_Impuls                := "M 4.2 Imp Cycle 0,4-sec",
           in_Impulszeit_in_100ms   := 4,
           in_Verzoegerungsart      := B#16#41,
           in_Verzoegerungszeit     := #Verz_Abgleich,
           io_Ausgangssignal        := #Ausgang_Timer,
           io_Zeitzaehler           := #Zeitzaehler);
NETWORK
TITLE = MemoryDruck nachführen
      A     #Ausgang_Timer;
      JC    NOPA;	//NO Pressure Adaptation
      L     #AbsolutDruck;
      T     #MemoryDruck;
NETWORK
TITLE = Relativdruck berechnen
NOPA: L     #AbsolutDruck;	//NO Pressure Adaptation
      L     #MemoryDruck;
      -R;
      T     #RelativDruck;
NETWORK
TITLE = Min-/Leer-/Maxdruck Druckfoerderung
      O(;
      L     #Auswahl_S_D;
      L     'D';
      <>I;
      );
      ON    #FRG_Druckstoerung;
      JC    SUFE;	//SUction FEeding
      A(;
      L     #RelativDruck;
      L     #MaxDruck;
      >=R;
      );
      A     #Geblaese_aktiv;
      A     #FRG_Druckstoerung;
      O     #Drahtbruch;
      S     #Druckstoerung;
      A(;
      L     #RelativDruck;
      L     #MinDruck;
      <=R;
      );
      AN    #Drahtbruch;
      R     #Druckstoerung;
      L     #RelativDruck;
      L     #LeerDruck;
      <=R;
      A     #FRG_Druckstoerung;
      AN    #Drahtbruch;
      =     #Leerdruck_aktiv;
NETWORK
TITLE = Min-/Maxdruck Saugfoerderung
SUFE: O(;	//SUction FEeding
      L     #Auswahl_S_D;
      L     'S';
      <>I;
      );
      ON    #FRG_Druckstoerung;
      JC    ENDF;	//END of Function
      A(;
      L     #RelativDruck;
      L     #MaxDruck;
      <=R;
      );
      A     #Geblaese_aktiv;
      A     #FRG_Druckstoerung;
      O     #Drahtbruch;
      S     #Druckstoerung;
      A(;
      L     #RelativDruck;
      L     #MinDruck;
      >=R;
      );
      AN    #Drahtbruch;
      R     #Druckstoerung;
      L     #RelativDruck;
      L     #LeerDruck;
      >=R;
      A     #FRG_Druckstoerung;
      AN    #Drahtbruch;
      =     #Leerdruck_aktiv;
NETWORK
TITLE = End of Function
ENDF: ON    #FRG_Druckstoerung;
      R     #Druckstoerung;
END_FUNCTION

FUNCTION "FC13 Standard Signals" : VOID	// FC 13
TITLE = Baustein für Standardmerker
//Erstellung:
//Datum        Bearbeiter                                                 Version
//--------------------------------------------------------------------------------
//26.06.97     R.Schaffert (sra)                                          01.00.00
//
//Änderungen:
//Nr. Datum    Bearb Änderung                                       Marke  Version
//--------------------------------------------------------------------------------
//01  21.11.02 sra   Resetmerker eingefügt                          (001) 01.00.01
//02  30.08.12 pti   Lampe Steuerspannung ein eingefügt             (002) 01.01.00
//03  23.07.13 sra   Signale für Sicherung eingefügt                (003) 01.02.00
//04  05.12.13 sra   Signal Steuerspannung gelöscht                       01.03.00
//05  02.06.14 sra   M0.3 Reset ebenfalls gelöscht (zu Änderung 04)       01.03.01
//06  14.12.16 sra   Implement SFC51 to read battery information    (006) 01.04.00
//________________________________________________________________________________
//Funktion:
//  
//Der Baustein erzeugt folgende Standardsignale:
//- M 0.1 "konstant 1" Merker
//- M 0.2 "konstant 0" Merker
//- M 1.6 Melderentprelltakt (5 Sekunden) 
//- M 1.7 "Takt Timernachbildung" = in_Basistakt_Timer
//- MB4 Impulsmerker für Takte 2.0s, 1.6s, 1.0s, 0.8s, 0.5s, 0.4s, 0.2s, 0.1s
//  !!! MB 2 muss als Taktmerker in CPU parametriert werden  !!
//  Das MB 3 wird als Hilfsbyte zur Flankenauswertung benutzt
//- MW 6 Zeitwert Takt = in_Zeit_Basistakt_100ms
AUTHOR : sra
FAMILY : AZO
VERSION : 0.0
VAR_INPUT
  in_E_Sicherung_OK : BOOL ;	//Eingang Sicherung OK = Eingang Störung Sicherung
  in_Basistakt_Timer : BOOL ;	//Taktmerker für alle Zeitfunktionen (abhängig von Zykluszeit)
  in_Zeit_Basistakt_100ms : INT ;	//Zeitwert Basistakt in 100 ms
END_VAR
VAR_OUTPUT
  o_Lampe_Stoer_Sicherung : BOOL ;	//Ausgang der Lampe "Störung Sicherung"
  o_Stoerung_Sicherung : BOOL ;	//Störung Sicherung -> für Störbitzuweisung im DB34
END_VAR
VAR_TEMP
  NOP : INT ;
END_VAR
BEGIN
NETWORK
TITLE = Statische Merker  
      SET;
      S     "M 0.1 Constant 1";
      R     "M 0.2 Constant 0";
NETWORK
TITLE = Lampe "Störung Sicherung" und Störmeldung Sicherung
//(003)
      AN    #in_E_Sicherung_OK;
      =     #o_Lampe_Stoer_Sicherung;
      =     #o_Stoerung_Sicherung;
NETWORK
TITLE = Impulsmerker Takte
//Impulsmerker für Takte 2.0s, 1.6s, 1.0s, 0.8s, 0.5s, 0.4s, 0.2s, 0.1s
//positive Flankenauswertung auf die von der CPU erzeugten Takte
      L     "MB 3 Edge Flags MB2";
      L     "MB 2 Cycle Flags";
      T     "MB 3 Edge Flags MB2";
      XOW;
      L     "MB 2 Cycle Flags";
      AW;
      T     "MB 4 Pulse Flags MB2";
NETWORK
TITLE = Werte für Timernachbildung vorgeben
//!! Abhängig von Zykluszeit !! 
      A     #in_Basistakt_Timer;
      =     "M 1.7 Cycle Timer-FC";
      L     #in_Zeit_Basistakt_100ms;
      T     "MW 6 Timer Val Cycle FCs";
NETWORK
TITLE = Takt Melderentprellung
//Takt Melderentprellung
      AN    "M 1.6 ClckDdebounceIndic";
      L     S5T#5S;
      SD    T 1;
      A     T 1;
      =     "M 1.6 ClckDdebounceIndic";
NETWORK
TITLE = read Battery fault of CPU
//(006)
      CALL  "RDSYSST" (
           REQ                      := "M 2.7 Cycle 2,0-sec",
           SZL_ID                   := W#16#392,
           INDEX                    := W#16#0,
           RET_VAL                  := "DB3 global Info".RDSYSST.RETVAL,
           BUSY                     := "DB3 global Info".RDSYSST.BUSY,
           SZL_HEADER               := "DB3 global Info".RDSYSST.SLZ_HEADER,
           DR                       := "DB3 global Info".RDSYSST.DR);	// W#16#392 = Status of the backup batteries in a rack/module rack of a CPU after at least one battery has failed /  if ID = 392h -> Index is always 0
      L     "DB3 global Info".RDSYSST.DR.Data_1;
      L     0;
      <>I;
      =     "DB3 global Info".Fehler_OB_Info.Battery_fault;
END_FUNCTION

FUNCTION "FC14 Debounce Indicator" : VOID	// FC 14
TITLE = Entprellung Füllstandsmelder
//Erstellung:
//Datum        Bearbeiter                                                 Version
//--------------------------------------------------------------------------------
//16.01.99     R.Schaffert (sra)                                          01.00.00
//
//Änderungen:
//Nr. Datum    Bearb Beschreibung                                   Marke Version
//--------------------------------------------------------------------------------
//01  
//
//________________________________________________________________________________
//Beschreibung: 
//
//Der Baustein entprellt den Signaleingang eines Melders. 
//
//Das Signal "Eingang enprellt" nimmt erst dann den Zustand des Signals "Eingang" 
//an, wenn über die Dauer von 2 Takten (Eingang  "Takt") der Zusatand des Signals 
//"Eingang" dauerhaft ungleich dem Signal "Eingang entprellt" ist.
//
AUTHOR : sra
FAMILY : AZO
VERSION : 0.0
VAR_INPUT
  Eingang : BOOL ;	//Eingangssignal des Melderes
  Takt : BOOL ;	//Taktsignal (Impulssignal)
END_VAR
VAR_IN_OUT
  Folgemerker : BOOL ;	//Hilfsmerker zum entprellen des Einganges
  Eingang_entprellt : BOOL ;	//Eingangssignal entprellt
END_VAR
VAR_TEMP
  Zwischenspeicher : BOOL ;
END_VAR
BEGIN
NETWORK
TITLE = Auswertung bei Taktpause
//Auswertung wenn Taktimpuls nicht ansteht
//
      A     #Takt;
      JC    Imp;
      AN    #Eingang;
      A     #Folgemerker;
      AN    #Eingang_entprellt;
      O;
      A     #Eingang;
      A     #Folgemerker;
      A     #Eingang_entprellt;
      R     #Folgemerker;
      JU    Ende;
NETWORK
TITLE = Auswertung bei Taktimpuls
//Auswertung wenn Taktimpuls ansteht
Imp:  A     #Eingang;
      A     #Folgemerker;
      S     #Eingang_entprellt;
      AN    #Eingang;
      A     #Folgemerker;
      R     #Eingang_entprellt;
      A     #Eingang;
      AN    #Eingang_entprellt;
      O;
      AN    #Eingang;
      A     #Eingang_entprellt;
      =     #Folgemerker;
Ende: NOP   0;
END_FUNCTION

FUNCTION "FC16 Fault evaluation" : VOID	// FC 16
TITLE = Sammelstoerung
//Erstellung:
//Datum        Bearbeiter                                                 Version
//--------------------------------------------------------------------------------
//26.07.99     M.Junker (jm)                                              01.00.00
//
//Änderungen:
//Nr. Datum    Bearb Änderung                                       Marke  Version
//--------------------------------------------------------------------------------
//01  14.09.99 jm    Spiegelung von PC ergänzt                            01.01.00
//02  06.10.99 jm    Störauswertung DWORD-weise                           01.02.00
//03  23.10.99 jm    QuitierungsDWORD von PC löschen                      01.03.00
//04  03.11.99 jm    Fehlerbeseitigung: QIP und DWORD                     01.03.01
//05  27.03.00 jm    Fehlerbeseitigung DWORD (Erstmeldung)                01.03.02
//06  19.04.05 jm    Fehlerbeseitigung Pointeradressen >8192(=>SLD) (006) 01.03.03
//07  23.02.06 jm    Quittierungs-DB Farbgrafik ist extern
//                   => Quittierung üder Kastor oder Farbgrafik     (007) 01.04.00
//08  23.03.06 sra   Einzelstörungsbereiche
//                   +Quitt.Erstwertmeldung über Quittierbereich         
//                   +Erstwertmeldung löschen ohne Störung          (008) 01.05.00
//09  10.05.06 sra   Fehlerbeseitigung zu Änderung 08               (009) 01.05.01
//10  11.05.06 sra   Änderung Quittierung von Farbgrafik            (010) 01.05.02
//11  05.10.06 jm    Anpassung für Siemens OP: extra Quittierbereich
//                   mit Flankenauswertung                          (011) 01.06.00
//12  01.04.08 jm    Steuerspannung entfernt, da Probleme mit OP-
//                   Quittierung (Problem: vorhandene Störung bei
//                   Steuerspannung aus am OP quittieren)           (012) 01.06.01
//13  16.11.15 sra   "Steuerspannung" in "Frg. Sammenstörung" geänd.(013) 01.06.02
//________________________________________________________________________________
//Beschreibung:
//
//!!!ACHTUNG: Parameter Anzahl Störungsbyte muß immer durch 4 teilbar sein!!!!
//
//Der Baustein überwacht einen definierbaren Teil eines Datenbaustein (DB34) in 
//dem alle Störmeldungen gesammelt werden. Sobald eine Störung vorhanden ist wird 
//das Signal "Sammelstörung" gebildet um damit z.B. eine Sammelstörlampe 
//anzusteuern. Der Parameter "Anzahl Störungsbyte" muß immer durch 4 teilbar sein
//
//In weiteren Bereichen weden die Datenblöcke "Erstmeldung", "Erstmeldung PC" und 
//Quittierung PC" mit der gleichen Größe wie der Störbereich benötigt.
//
//Funktion:
//Um bei der Störungsquittierung zur FG kompatibel zu sein werden die 
//Quittierungen, sobald die Störung verschwunden ist, von der SPS gelöscht.
//
//Die beiden Quittierungsbereiche (in DB34 für Kastor; in DB35 für SCADA) werden 
//mit ODER ausgewertet, d.h. die Störungen könnten von beiden Seiten quittiert 
//werden (wird normal nicht gemacht). Die Quittierbits werden hier so umkopiert, 
//daß sie immer in beiden Quittierungsbereichen auftauchen.
//=> es müssen immer beide Quittierbereiche angelegt sein
//=> an den Aggregat-Baustein werden die Bits aus dem DB35 angelegt
//
//OP:
//Siemens OPs müssen in einen extra Bereich quittieren, der hinter dem normalen 
//Standardbereichen im DB34 liegt. Im Anschluss folgt noch ein Bereich für die 
//Flankenauswertung. Bei positiver Flanke der Quittierung von OP wird die in den 
//Bereich der SCADA-Quittierung übertragen. In den OP Quittierbereich darf auf 
//gar keinen Fall die SPS schreiben. Wird kein OP verwendet so können die 
//OP-Bereiche aus dem DB34 weggelassen werden.
AUTHOR : jm
FAMILY : STANDARD
NAME : hsh
VERSION : 0.0
VAR_INPUT
  Conf_AckBySiemensOP : BOOL ;	//configuration bit: ackowledge done by Siemens OP (011)
  Stoerungstakt : BOOL ;	//Takt für Störauswertung
  Freigabe_Sammelstoerung : BOOL ;	//Freigabe Sammelstörung (ehemals Steuerspannung)
  Quittierung : BOOL ;	//Quittierung Fehlermeldung
  Stoerungs_DB : INT ;	//Stör-Datenbaustein
  Quittierungs_DB_SCADA : INT ;	//Quittier-Datenbaustein Farbgrafik
  Anzahl_Stoerungs_Byte : INT ;	//Anzahl Störungsbyte im Stör-Db (Blocklänge der 4 Bereiche)
  Offset_Stoerungs_Byte : INT ;	//Anfangs-DW der Störmeldungen im Stör-DB (wenn Bereich nicht bei Byte 0 anfängt)
  Adresse_Anfangswort : INT ;	//Adresse des ersten Datenwortes das ausgewertet wird
  Bereichslaenge : INT ;	//Länge des Bereiches der ausgewertet wird (!!Muss durch 4 teilbar sein!!)
END_VAR
VAR_IN_OUT
  Sammelstoerung : BOOL ;	//Sammelstörung
  Erstmeldung : BOOL ;	//Erstmeldung aktiv
  Erstmeldung_PC : BOOL ;	//Erstmeldung an PC
  Quittierung_PC : BOOL ;	//Quittierung von PC
END_VAR
VAR_TEMP
  Stoer_DB : INT ;	//Stoerungs-DB lokal
  Quit_DB : INT ;	//Quittierungs-DB extern
  Offsetende : INT ;	//= Störungsbyte + Offset
  SI : INT ;	//Störungsindex
  KI : INT ;	//Kopierindex
  SIP : INT ;	//Spiegelungsindex PC
  QIP : INT ;	//Quittierungsindex PC
  QIS : INT ;	//Quitierungsindex SCADA
  QIO : INT ;	//Quittierungsindex Siemens OP (011)
  KQIO : INT ;	//Kopie Quittierungsindex Siemens OP (011)
  StoerungsDWORD : DWORD ;	//Stoerungsdoppelwort
  KopieDWORD : DWORD ;	//Kopiedoppelwort
  SpiegelungsDWORD : DWORD ;	//Spiegelungsdoppelwort
  QuittierungsDWORD : DWORD ;	//Quittierungsdoppelwort
  QuitPC_DWORD : DWORD ;	//Quittierungsdoppelwort von PC
  QuitSCADA_DWORD : DWORD ;	//Quittierungsdoppelwort von SCADA
  QuitOP_DWORD : DWORD ;	//Quittierungdoppelwort von OP (011)
  KopieQuitOP_DWORD : DWORD ;	//Kopie Quittierungdoppelwort von OP (011)
  t_Erstmeldung_PC : BOOL ;	//Erstmeldung an PC
END_VAR
BEGIN
NETWORK
TITLE = Störauswertung aktiv?
//      ON    #Steuerspannung // (012)
//      SPB   FCEN                       // FunCtion ENd // (012)
      ON    #Stoerungstakt;
      JC    QUIT;	// QUITtierung Erstmeldung prüfen
NETWORK
TITLE = Variablen vorbelegen
//Minus 4 wegen DWORD-Auswertung
      CLR;
      =     #Sammelstoerung;
      =     #t_Erstmeldung_PC;
      L     #Offset_Stoerungs_Byte;
      L     #Adresse_Anfangswort;	// (008)
      +I;	// (008)
      L     #Bereichslaenge;	// (008)
      +I;
      T     #Offsetende;	//Offsetende = Offset + Anzahl // (007)
      L     #Offsetende;	// (007)
      L     4;
      -I;
      T     #SI;	//Stoerungsindex = Offsetende + Anzahl -4
      T     #QIS;	//Quittierungsindex SCADA = Stoerungsindex (007)
      L     #Offsetende;	// (007)
      L     #Anzahl_Stoerungs_Byte;	// (008)
      +I;
      L     4;
      -I;
      T     #KI;	//Kopierindex = Offsetende + Anzahl*2 -4
      L     #Offsetende;	// (007)
      L     #Anzahl_Stoerungs_Byte;
      +I;
      L     #Anzahl_Stoerungs_Byte;	// (008)
      +I;
      L     4;
      -I;
      T     #SIP;	//Spiegelungsindex PC = Offsetende + Anzahl*3 -4
      L     #Offsetende;	// (007)
      L     #Anzahl_Stoerungs_Byte;
      +I;
      L     #Anzahl_Stoerungs_Byte;
      +I;
      L     #Anzahl_Stoerungs_Byte;	// (008)
      +I;
      L     4;
      -I;
      T     #QIP;	//Quittierungsindex PC = Offsetende + Anzahl*4 -4
// >>>>>>>>>> (011)
      L     #Offsetende;
      L     #Anzahl_Stoerungs_Byte;
      +I;
      L     #Anzahl_Stoerungs_Byte;
      +I;
      L     #Anzahl_Stoerungs_Byte;
      +I;
      L     #Anzahl_Stoerungs_Byte;
      +I;
      L     4;
      -I;
      T     #QIO;	//Quittierungsindex OP = Offsetende + Anzahl*5 -4
      L     #Offsetende;
      L     #Anzahl_Stoerungs_Byte;
      +I;
      L     #Anzahl_Stoerungs_Byte;
      +I;
      L     #Anzahl_Stoerungs_Byte;
      +I;
      L     #Anzahl_Stoerungs_Byte;
      +I;
      L     #Anzahl_Stoerungs_Byte;
      +I;
      L     4;
      -I;
      T     #KQIO;	//Kopie Quittierungsindex OP = Offsetende + Anzahl*6 -4
// <<<<<<<<<< (011)
NETWORK
TITLE = Störungs-/Kopie-/Spiegelungs-/QuittierungsDWORD(OP) laden
      L     #Stoerungs_DB;
      T     #Stoer_DB;
      L     #Quittierungs_DB_SCADA;	// (007)
      T     #Quit_DB;	// (007)
SLOP: OPN   DB [#Stoer_DB];
      L     #SI;
      SLD   3;	// (006)
      LAR1;
      L     DBD [AR1,P#0.0];
      T     #StoerungsDWORD;
      L     #KI;
      SLD   3;	// (006)
      LAR1;
      L     DBD [AR1,P#0.0];
      T     #KopieDWORD;
      L     #SIP;
      SLD   3;	// (006)
      LAR1;
      L     DBD [AR1,P#0.0];
      T     #SpiegelungsDWORD;
      L     #QIP;
      SLD   3;	// (006)
      LAR1;
      L     DBD [AR1,P#0.0];
      T     #QuitPC_DWORD;	// (007)
///*(007)
      L     L#0;	// (011)
      T     #QuitSCADA_DWORD;
      L     #Quittierungs_DB_SCADA;	// (011)
      L     0;
      ==I;	// (011)
      JC    KQ1;	// (011) kein Quittierungsbaustein vorhanden
      OPN   DB [#Quit_DB];
      L     #QIS;
      SLD   3;
      LAR1;
      L     DBD [AR1,P#0.0];
      T     #QuitSCADA_DWORD;
      OPN   DB [#Stoer_DB];
//(007)*/
// >>>>>>>>>> (011)
      L     0;
      T     #QuitOP_DWORD;	// vorbelegen, falls nicht vorhanden
      AN    #Conf_AckBySiemensOP;
      JC    NOPA;	// No OP Acknowledge
      L     #QIO;
      SLD   3;
      LAR1;
      L     DBD [AR1,P#0.0];
      T     #QuitOP_DWORD;
      L     #KQIO;
      SLD   3;
      LAR1;
      L     DBD [AR1,P#0.0];
      T     #KopieQuitOP_DWORD;
NOPA: NOP   0;	// No OP Acknowledge
// <<<<<<<<<< (011)
KQ1:  NOP   0;
NETWORK
TITLE = Pos.Flanke Quittierung OP
//(011)
      AN    #Conf_AckBySiemensOP;
      JC    NPOA;	// No Processing of Op Acknowledge
      L     #QuitOP_DWORD;	// -
      L     #KopieQuitOP_DWORD;	// |
      XOD;	// | positive Flanke Quittierung OP
      L     #QuitOP_DWORD;	// |
      AD;	// -
      L     #QuitSCADA_DWORD;
      OD;
      T     #QuitSCADA_DWORD;	// => Quittierung in QuitSCADA setzen
      L     #QuitOP_DWORD;
      T     #KopieQuitOP_DWORD;	// => Hilfsmerker Flanke (Kopie ALT)
NETWORK
TITLE = Quittierung OP DWORD nach Kopiebyte
//(011)
      L     #KQIO;
      SLD   3;
      LAR1;
      L     #KopieQuitOP_DWORD;
      T     DBD [AR1,P#0.0];	// => Quittierung OP merken
NPOA: NOP   0;
NETWORK
TITLE = Sammelstörung
      L     #StoerungsDWORD;
      L     0;
      <>D;
      A     #Freigabe_Sammelstoerung;	// (012)
      S     #Sammelstoerung;
NETWORK
TITLE = Erstwertmeldung
      L     #StoerungsDWORD;
      L     #KopieDWORD;
      XOD;
      L     #StoerungsDWORD;
      AD;
      L     0;
      <>D;
      A     #Freigabe_Sammelstoerung;	// (012)
      S     #Erstmeldung;
NETWORK
TITLE = Erstwertmeldung an PC
      L     #StoerungsDWORD;
      L     #SpiegelungsDWORD;
      <>D;
      S     #t_Erstmeldung_PC;
NETWORK
TITLE = StoerungsDWORD nach Kopiebyte
      L     #KI;
      SLD   3;	// (006)
      LAR1;
      L     #StoerungsDWORD;
      T     DBD [AR1,P#0.0];
NETWORK
TITLE = neue Quittierung?
//(008)
      L     #QuitSCADA_DWORD;
      L     #QuitPC_DWORD;
      XOD;
      L     0;
      <>D;
      R     #Erstmeldung;
NETWORK
TITLE = QuittierungsDWORD bilden
//(007)
      L     #QuitPC_DWORD;	// (010)
      L     #SpiegelungsDWORD;	// (010)
      AD;	// (010)
      L     #QuitSCADA_DWORD;
      OD;
      T     #QuittierungsDWORD;	// Quittierung von Kastor oder SCADA
NETWORK
TITLE = QuittierungsDWORD löschen
      L     #StoerungsDWORD;
      L     #QuittierungsDWORD;
      AD;
      T     #QuittierungsDWORD;
NETWORK
TITLE = QuittierungsDWORD PC und SCADA löschen
      L     #QIP;
      SLD   3;	// (006)
      LAR1;
      L     #QuittierungsDWORD;
      T     DBD [AR1,P#0.0];	// PC Quittierung
      L     #Quittierungs_DB_SCADA;	// (011)
      L     0;	// (011)
      ==I;	// (011)
      JC    KQ2;	// (011) kein Quittierungsbaustein vorhanden
///*(007)
      OPN   DB [#Quit_DB];
      L     #QIS;
      SLD   3;
      LAR1;
      L     #QuittierungsDWORD;
      T     DBD [AR1,P#0.0];	// SCADA Quittierung
//(007)*/
KQ2:  NOP   0;
NETWORK
TITLE = Störungsschleife von (Anzahl - 4) bis 0
//Minus 4 wegen DWORD-Auswertung
// >>>>>>>>>> (011)
      L     #KQIO;
      L     4;
      -I;
      T     #KQIO;
      L     #QIO;
      L     4;
      -I;
      T     #QIO;
// <<<<<<<<<< (011)
///*(007)
      L     #QIS;
      L     4;
      -I;
      T     #QIS;
//(007)*/
      L     #QIP;
      L     4;
      -I;
      T     #QIP;
      L     #SIP;
      L     4;
      -I;
      T     #SIP;
      L     #KI;
      L     4;
      -I;
      T     #KI;
      L     #SI;
      L     4;
      -I;
      T     #SI;
      L     #Offset_Stoerungs_Byte;
      L     #Adresse_Anfangswort;	// (008)
      +I;	// (008)
      L     #SI;	// (008)
      <=I;	// (008) (009)
      JC    SLOP;	// Störungs LOOP
NETWORK
TITLE = Störauswertung für PC aktiv?
      O     #Erstmeldung_PC;
      O     #Quittierung_PC;
      JC    QUIT;	//QUITtierung
      A     #t_Erstmeldung_PC;
      S     #Erstmeldung_PC;
NETWORK
TITLE = Erstmeldung quittiert?
QUIT: A     #Quittierung;	//QUITtierung
      ON    #Sammelstoerung;	// (008)
      R     #Erstmeldung;
      A     #Quittierung_PC;
      R     #Erstmeldung_PC;
      NOP   0;
END_FUNCTION

